LIN {X -0.155,Y -578.900,Z 921.405,A 0.000,B 0.000,C 90.000,E1 108.852} C_DIS
LIN {X -0.107,Y -571.910,Z 921.403,A 0.000,B 0.000,C 90.000,E1 108.471} C_DIS
LIN {X 0.202,Y -564.890,Z 921.401,A 0.000,B 0.000,C 90.000,E1 108.127} C_DIS
LIN {X -0.065,Y -557.655,Z 921.399,A 0.000,B 0.000,C 90.000,E1 107.873} C_DIS
LIN {X -0.326,Y -554.957,Z 921.399,A 0.000,B 0.000,C 90.000,E1 107.764} C_DIS
LIN {X -0.045,Y -553.341,Z 921.398,A 0.000,B 0.000,C 90.000,E1 107.583} C_DIS
LIN {X -0.084,Y -553.320,Z 921.398,A 0.000,B 0.000,C 90.000,E1 107.583} C_DIS
LIN {X 0.080,Y -552.969,Z 921.396,A 0.000,B 0.000,C 90.000,E1 107.347} C_DIS
LIN {X 0.102,Y -553.748,Z 921.385,A 0.000,B 0.000,C 90.000,E1 105.245} C_DIS
LIN {X 0.147,Y -554.848,Z 921.372,A 0.000,B 0.000,C 90.000,E1 103.008} C_DIS
LIN {X -0.166,Y -556.747,Z 921.357,A 0.000,B 0.000,C 90.000,E1 100.254} C_DIS
LIN {X -0.129,Y -557.796,Z 921.349,A 0.000,B 0.000,C 90.000,E1 98.859} C_DIS
LIN {X -0.015,Y -558.994,Z 921.340,A 0.000,B 0.000,C 90.000,E1 97.182} C_DIS
LIN {X -0.155,Y -559.710,Z 921.334,A 0.000,B 0.000,C 90.000,E1 96.087} C_DIS
LIN {X -0.153,Y -560.546,Z 921.326,A 0.000,B 0.000,C 90.000,E1 94.702} C_DIS
LIN {X -0.229,Y -561.254,Z 921.318,A 0.000,B 0.000,C 90.000,E1 93.326} C_DIS
LIN {X -0.283,Y -561.918,Z 921.311,A 0.000,B 0.000,C 90.000,E1 91.949} C_DIS
LIN {X 0.131,Y -562.359,Z 921.305,A 0.000,B 0.000,C 90.000,E1 90.802} C_DIS
LIN {X 0.078,Y -562.761,Z 921.297,A 0.000,B 0.000,C 90.000,E1 89.427} C_DIS
LIN {X -0.075,Y -562.990,Z 921.291,A 0.000,B 0.000,C 90.000,E1 88.339} C_DIS
LIN {X 0.023,Y -563.336,Z 921.282,A 0.000,B 0.000,C 90.000,E1 86.674} C_DIS
LIN {X 0.137,Y -563.594,Z 921.272,A 0.000,B 0.000,C 90.000,E1 85.008} C_DIS
LIN {X -0.167,Y -563.962,Z 921.262,A 0.000,B 0.000,C 90.000,E1 83.109} C_DIS
LIN {X 0.070,Y -564.278,Z 921.253,A 0.000,B 0.000,C 90.000,E1 81.432} C_DIS
LIN {X 0.014,Y -564.989,Z 921.242,A 0.000,B 0.000,C 90.000,E1 79.511} C_DIS
LIN {X -0.025,Y -565.940,Z 921.231,A 0.000,B 0.000,C 90.000,E1 77.589} C_DIS
LIN {X 0.193,Y -567.056,Z 921.220,A 0.000,B 0.000,C 90.000,E1 75.644} C_DIS
LIN {X -0.131,Y -568.000,Z 921.211,A 0.000,B 0.000,C 90.000,E1 74.031} C_DIS
LIN {X 0.112,Y -568.779,Z 921.202,A 0.000,B 0.000,C 90.000,E1 72.362} C_DIS
LIN {X 0.340,Y -569.551,Z 921.191,A 0.000,B 0.000,C 90.000,E1 70.423} C_DIS
LIN {X -0.267,Y -569.891,Z 921.185,A 0.000,B 0.000,C 90.000,E1 69.390} C_DIS
LIN {X 0.036,Y -570.321,Z 921.176,A 0.000,B 0.000,C 90.000,E1 67.720} C_DIS
LIN {X -0.005,Y -570.513,Z 921.169,A 0.000,B 0.000,C 90.000,E1 66.357} C_DIS
LIN {X 0.014,Y -570.742,Z 921.160,A 0.000,B 0.000,C 90.000,E1 64.717} C_DIS
LIN {X 0.198,Y -570.867,Z 921.152,A 0.000,B 0.000,C 90.000,E1 63.332} C_DIS
LIN {X -0.048,Y -570.821,Z 921.143,A 0.000,B 0.000,C 90.000,E1 61.719} C_DIS
LIN {X 0.151,Y -570.814,Z 921.135,A 0.000,B 0.000,C 90.000,E1 60.333} C_DIS
LIN {X 0.036,Y -570.701,Z 921.129,A 0.000,B 0.000,C 90.000,E1 59.253} C_DIS
LIN {X -0.373,Y -570.505,Z 921.123,A 0.000,B 0.000,C 90.000,E1 58.201} C_DIS
LIN {X 0.296,Y -570.066,Z 921.117,A 0.000,B 0.000,C 90.000,E1 57.041} C_DIS
LIN {X 0.167,Y -569.577,Z 921.111,A 0.000,B 0.000,C 90.000,E1 55.960} C_DIS
LIN {X -0.248,Y -569.113,Z 921.107,A 0.000,B 0.000,C 90.000,E1 55.182} C_DIS
LIN {X 0.131,Y -568.532,Z 921.102,A 0.000,B 0.000,C 90.000,E1 54.322} C_DIS
LIN {X 0.171,Y -567.857,Z 921.097,A 0.000,B 0.000,C 90.000,E1 53.497} C_DIS
LIN {X 0.205,Y -566.668,Z 921.091,A 0.000,B 0.000,C 90.000,E1 52.396} C_DIS
LIN {X -0.123,Y -565.340,Z 921.085,A 0.000,B 0.000,C 90.000,E1 51.331} C_DIS
LIN {X 0.235,Y -563.649,Z 921.079,A 0.000,B 0.000,C 90.000,E1 50.194} C_DIS
LIN {X 0.111,Y -562.253,Z 921.074,A 0.000,B 0.000,C 90.000,E1 49.380} C_DIS
LIN {X -0.033,Y -560.643,Z 921.070,A 0.000,B 0.000,C 90.000,E1 48.566} C_DIS
LIN {X 0.176,Y -558.833,Z 921.065,A 0.000,B 0.000,C 90.000,E1 47.715} C_DIS
LIN {X 0.294,Y -557.537,Z 921.062,A 0.000,B 0.000,C 90.000,E1 47.148} C_DIS
LIN {X 0.124,Y -554.396,Z 921.056,A 0.000,B 0.000,C 90.000,E1 46.053} C_DIS
LIN {X -0.220,Y -553.596,Z 921.054,A 0.000,B 0.000,C 90.000,E1 45.810} C_DIS
LIN {X 0.294,Y -550.777,Z 921.050,A 0.000,B 0.000,C 90.000,E1 44.919} C_DIS
LIN {X -0.033,Y -548.775,Z 921.047,A 0.000,B 0.000,C 90.000,E1 44.393} C_DIS
LIN {X 0.042,Y -545.409,Z 921.042,A 0.000,B 0.000,C 90.000,E1 43.542} C_DIS
LIN {X 0.065,Y -543.005,Z 921.039,A 0.000,B 0.000,C 90.000,E1 42.975} C_DIS
LIN {X 0.081,Y -537.557,Z 921.033,A 0.000,B 0.000,C 90.000,E1 41.838} C_DIS
LIN {X -0.142,Y -533.753,Z 921.029,A 0.000,B 0.000,C 90.000,E1 41.148} C_DIS
LIN {X 0.007,Y -529.606,Z 921.025,A 0.000,B 0.000,C 90.000,E1 40.415} C_DIS
LIN {X -0.131,Y -524.206,Z 921.020,A 0.000,B 0.000,C 90.000,E1 39.564} C_DIS
LIN {X 0.068,Y -518.435,Z 921.015,A 0.000,B 0.000,C 90.000,E1 38.669} C_DIS
LIN {X 0.073,Y -513.345,Z 921.011,A 0.000,B 0.000,C 90.000,E1 37.935} C_DIS
LIN {X -0.276,Y -508.013,Z 921.007,A 0.000,B 0.000,C 90.000,E1 37.237} C_DIS
LIN {X 0.134,Y -500.920,Z 921.002,A 0.000,B 0.000,C 90.000,E1 36.297} C_DIS
LIN {X -0.105,Y -495.831,Z 920.998,A 0.000,B 0.000,C 90.000,E1 35.724} C_DIS
LIN {X 0.138,Y -490.507,Z 920.995,A 0.000,B 0.000,C 90.000,E1 35.105} C_DIS
LIN {X 0.216,Y -483.823,Z 920.991,A 0.000,B 0.000,C 90.000,E1 34.405} C_DIS
LIN {X 0.006,Y -477.975,Z 920.988,A 0.000,B 0.000,C 90.000,E1 33.865} C_DIS
LIN {X 0.120,Y -469.147,Z 920.984,A 0.000,B 0.000,C 90.000,E1 33.038} C_DIS
LIN {X -0.025,Y -460.160,Z 920.979,A 0.000,B 0.000,C 90.000,E1 32.260} C_DIS
LIN {X 0.081,Y -447.901,Z 920.974,A 0.000,B 0.000,C 90.000,E1 31.209} C_DIS
LIN {X 0.065,Y -430.957,Z 920.966,A 0.000,B 0.000,C 90.000,E1 29.795} C_DIS
LIN {X 0.023,Y -409.707,Z 920.955,A 0.000,B 0.000,C 90.000,E1 27.897} C_DIS
LIN {X -0.106,Y -401.030,Z 920.950,A 0.000,B 0.000,C 90.000,E1 27.052} C_DIS
LIN {X -0.127,Y -395.925,Z 920.947,A 0.000,B 0.000,C 90.000,E1 26.488} C_DIS
LIN {X -0.007,Y -394.135,Z 920.946,A 0.000,B 0.000,C 90.000,E1 26.232} C_DIS
LIN {X -0.213,Y -392.254,Z 920.944,A 0.000,B 0.000,C 90.000,E1 25.976} C_DIS
LIN {X -0.062,Y -390.731,Z 920.942,A 0.000,B 0.000,C 90.000,E1 25.643} C_DIS
LIN {X -0.113,Y -389.363,Z 920.940,A 0.000,B 0.000,C 90.000,E1 25.155} C_DIS
LIN {X 0.064,Y -388.954,Z 920.939,A 0.000,B 0.000,C 90.000,E1 24.951} C_DIS
LIN {X 0.166,Y -388.518,Z 920.936,A 0.000,B 0.000,C 90.000,E1 24.387} C_DIS
LIN {X 0.058,Y -388.642,Z 920.932,A 0.000,B 0.000,C 90.000,E1 23.695} C_DIS
LIN {X -0.105,Y -392.840,Z 920.906,A 0.000,B 0.000,C 90.000,E1 19.087} C_DIS
LIN {X -0.142,Y -396.197,Z 920.890,A 0.000,B 0.000,C 90.000,E1 16.260} C_DIS
LIN {X 0.067,Y -400.345,Z 920.873,A 0.000,B 0.000,C 90.000,E1 13.063} C_DIS
LIN {X 0.165,Y -404.546,Z 920.857,A 0.000,B 0.000,C 90.000,E1 10.254} C_DIS
LIN {X -0.171,Y -408.566,Z 920.844,A 0.000,B 0.000,C 90.000,E1 7.871} C_DIS
LIN {X -0.138,Y -412.265,Z 920.832,A 0.000,B 0.000,C 90.000,E1 5.796} C_DIS
LIN {X -0.085,Y -415.633,Z 920.823,A 0.000,B 0.000,C 90.000,E1 4.073} C_DIS
LIN {X 0.178,Y -422.235,Z 920.806,A 0.000,B 0.000,C 90.000,E1 0.974} C_DIS
LIN {X 0.034,Y -429.232,Z 920.790,A 0.000,B 0.000,C 90.000,E1 358.108} C_DIS
LIN {X 0.171,Y -431.299,Z 920.786,A 0.000,B 0.000,C 90.000,E1 357.421} C_DIS
LIN {X -0.148,Y -433.347,Z 920.783,A 0.000,B 0.000,C 90.000,E1 356.963} C_DIS
LIN {X -0.112,Y -436.667,Z 920.780,A 0.000,B 0.000,C 90.000,E1 356.445} C_DIS
LIN {X -0.068,Y -438.404,Z 920.779,A 0.000,B 0.000,C 90.000,E1 356.274} C_DIS
LIN {X 0.123,Y -441.542,Z 920.778,A 0.000,B 0.000,C 90.000,E1 355.988} C_DIS
LIN {X 0.114,Y -447.681,Z 920.776,A 0.000,B 0.000,C 90.000,E1 355.641} C_DIS
LIN {X 0.084,Y -456.667,Z 920.774,A 0.000,B 0.000,C 90.000,E1 355.241} C_DIS
LIN {X 0.004,Y -466.607,Z 920.771,A 0.000,B 0.000,C 90.000,E1 354.780} C_DIS
LIN {X 0.197,Y -483.309,Z 920.766,A 0.000,B 0.000,C 90.000,E1 353.913} C_DIS
LIN {X 0.043,Y -493.230,Z 920.763,A 0.000,B 0.000,C 90.000,E1 353.394} C_DIS
LIN {X -0.231,Y -506.078,Z 920.759,A 0.000,B 0.000,C 90.000,E1 352.704} C_DIS
LIN {X -0.105,Y -515.398,Z 920.756,A 0.000,B 0.000,C 90.000,E1 352.129} C_DIS
LIN {X -0.100,Y -521.738,Z 920.754,A 0.000,B 0.000,C 90.000,E1 351.724} C_DIS
LIN {X -0.148,Y -530.798,Z 920.750,A 0.000,B 0.000,C 90.000,E1 351.084} C_DIS
LIN {X -0.007,Y -536.690,Z 920.748,A 0.000,B 0.000,C 90.000,E1 350.622} C_DIS
LIN {X -0.031,Y -544.823,Z 920.744,A 0.000,B 0.000,C 90.000,E1 349.926} C_DIS
LIN {X 0.170,Y -550.298,Z 920.741,A 0.000,B 0.000,C 90.000,E1 349.398} C_DIS
LIN {X 0.037,Y -556.664,Z 920.738,A 0.000,B 0.000,C 90.000,E1 348.757} C_DIS
LIN {X 0.139,Y -564.802,Z 920.732,A 0.000,B 0.000,C 90.000,E1 347.825} C_DIS
LIN {X -0.193,Y -570.375,Z 920.729,A 0.000,B 0.000,C 90.000,E1 347.173} C_DIS
LIN {X 0.286,Y -577.495,Z 920.723,A 0.000,B 0.000,C 90.000,E1 346.172} C_DIS
LIN {X 0.054,Y -582.153,Z 920.720,A 0.000,B 0.000,C 90.000,E1 345.519} C_DIS
LIN {X 0.018,Y -589.016,Z 920.714,A 0.000,B 0.000,C 90.000,E1 344.448} C_DIS
LIN {X 0.142,Y -594.307,Z 920.708,A 0.000,B 0.000,C 90.000,E1 343.504} C_DIS
LIN {X -0.310,Y -600.032,Z 920.703,A 0.000,B 0.000,C 90.000,E1 342.489} C_DIS
LIN {X -0.180,Y -603.379,Z 920.699,A 0.000,B 0.000,C 90.000,E1 341.819} C_DIS
LIN {X 0.250,Y -608.561,Z 920.693,A 0.000,B 0.000,C 90.000,E1 340.732} C_DIS
LIN {X -0.112,Y -611.757,Z 920.690,A 0.000,B 0.000,C 90.000,E1 340.115} C_DIS
LIN {X -0.151,Y -616.431,Z 920.684,A 0.000,B 0.000,C 90.000,E1 339.082} C_DIS
LIN {X 0.094,Y -620.959,Z 920.678,A 0.000,B 0.000,C 90.000,E1 338.028} C_DIS
LIN {X 0.163,Y -626.123,Z 920.671,A 0.000,B 0.000,C 90.000,E1 336.741} C_DIS
LIN {X -0.041,Y -629.861,Z 920.665,A 0.000,B 0.000,C 90.000,E1 335.741} C_DIS
LIN {X 0.147,Y -635.046,Z 920.657,A 0.000,B 0.000,C 90.000,E1 334.204} C_DIS
LIN {X 0.001,Y -637.559,Z 920.653,A 0.000,B 0.000,C 90.000,E1 333.461} C_DIS
LIN {X -0.230,Y -642.060,Z 920.644,A 0.000,B 0.000,C 90.000,E1 331.975} C_DIS
LIN {X -0.139,Y -645.370,Z 920.637,A 0.000,B 0.000,C 90.000,E1 330.717} C_DIS
LIN {X 0.015,Y -648.503,Z 920.630,A 0.000,B 0.000,C 90.000,E1 329.459} C_DIS
LIN {X 0.218,Y -651.364,Z 920.623,A 0.000,B 0.000,C 90.000,E1 328.201} C_DIS
LIN {X -0.187,Y -653.364,Z 920.618,A 0.000,B 0.000,C 90.000,E1 327.248} C_DIS
LIN {X 0.341,Y -655.077,Z 920.613,A 0.000,B 0.000,C 90.000,E1 326.215} C_DIS
LIN {X -0.099,Y -656.881,Z 920.606,A 0.000,B 0.000,C 90.000,E1 325.022} C_DIS
LIN {X 0.023,Y -658.426,Z 920.599,A 0.000,B 0.000,C 90.000,E1 323.783} C_DIS
LIN {X -0.025,Y -659.952,Z 920.591,A 0.000,B 0.000,C 90.000,E1 322.316} C_DIS
LIN {X -0.030,Y -661.230,Z 920.583,A 0.000,B 0.000,C 90.000,E1 320.848} C_DIS
LIN {X -0.018,Y -662.403,Z 920.574,A 0.000,B 0.000,C 90.000,E1 319.380} C_DIS
LIN {X -0.065,Y -664.772,Z 920.561,A 0.000,B 0.000,C 90.000,E1 316.944} C_DIS
LIN {X -0.090,Y -665.637,Z 920.555,A 0.000,B 0.000,C 90.000,E1 315.972} C_DIS
LIN {X -0.093,Y -667.802,Z 920.541,A 0.000,B 0.000,C 90.000,E1 313.299} C_DIS
LIN {X -0.035,Y -669.268,Z 920.532,A 0.000,B 0.000,C 90.000,E1 311.838} C_DIS
LIN {X 0.052,Y -670.558,Z 920.524,A 0.000,B 0.000,C 90.000,E1 310.378} C_DIS
LIN {X -0.280,Y -671.560,Z 920.518,A 0.000,B 0.000,C 90.000,E1 309.197} C_DIS
LIN {X 0.350,Y -672.330,Z 920.512,A 0.000,B 0.000,C 90.000,E1 308.177} C_DIS
LIN {X 0.169,Y -673.343,Z 920.504,A 0.000,B 0.000,C 90.000,E1 306.744} C_DIS
LIN {X 0.005,Y -673.961,Z 920.496,A 0.000,B 0.000,C 90.000,E1 305.311} C_DIS
LIN {X -0.143,Y -674.489,Z 920.490,A 0.000,B 0.000,C 90.000,E1 304.119} C_DIS
LIN {X 0.037,Y -675.372,Z 920.480,A 0.000,B 0.000,C 90.000,E1 302.418} C_DIS
LIN {X -0.170,Y -676.603,Z 920.469,A 0.000,B 0.000,C 90.000,E1 300.512} C_DIS
LIN {X 0.121,Y -680.212,Z 920.451,A 0.000,B 0.000,C 90.000,E1 297.129} C_DIS
LIN {X 0.232,Y -682.979,Z 920.440,A 0.000,B 0.000,C 90.000,E1 295.207} C_DIS
LIN {X 0.163,Y -684.330,Z 920.435,A 0.000,B 0.000,C 90.000,E1 294.259} C_DIS
LIN {X -0.104,Y -685.114,Z 920.431,A 0.000,B 0.000,C 90.000,E1 293.567} C_DIS
LIN {X 0.049,Y -685.476,Z 920.428,A 0.000,B 0.000,C 90.000,E1 293.078} C_DIS
LIN {X 0.210,Y -685.469,Z 920.426,A 0.000,B 0.000,C 90.000,E1 292.589} C_DIS
LIN {X -0.211,Y -685.321,Z 920.424,A 0.000,B 0.000,C 90.000,E1 292.386} C_DIS
LIN {X -0.049,Y -683.903,Z 920.422,A 0.000,B 0.000,C 90.000,E1 291.897} C_DIS
LIN {X -0.097,Y -682.936,Z 920.420,A 0.000,B 0.000,C 90.000,E1 291.663} C_DIS
LIN {X 0.005,Y -682.139,Z 920.420,A 0.000,B 0.000,C 90.000,E1 291.535} C_DIS
LIN {X 0.106,Y -680.957,Z 920.419,A 0.000,B 0.000,C 90.000,E1 291.408} C_DIS
LIN {X 0.061,Y -677.819,Z 920.418,A 0.000,B 0.000,C 90.000,E1 291.173} C_DIS
LIN {X -0.109,Y -676.090,Z 920.417,A 0.000,B 0.000,C 90.000,E1 291.046} C_DIS
LIN {X 0.122,Y -674.544,Z 920.416,A 0.000,B 0.000,C 90.000,E1 290.918} C_DIS
LIN {X -0.114,Y -662.599,Z 920.413,A 0.000,B 0.000,C 90.000,E1 290.301} C_DIS
LIN {X 0.133,Y -661.615,Z 920.412,A 0.000,B 0.000,C 90.000,E1 290.174} C_DIS
LIN {X 0.072,Y -661.583,Z 920.412,A 0.000,B 0.000,C 90.000,E1 290.174} C_DIS
LIN {X -0.280,Y -661.528,Z 920.411,A 0.000,B 0.000,C 90.000,E1 290.066} C_DIS
LIN {X -0.188,Y -661.993,Z 920.410,A 0.000,B 0.000,C 90.000,E1 289.812} C_DIS
LIN {X -0.296,Y -662.586,Z 920.409,A 0.000,B 0.000,C 90.000,E1 289.577} C_DIS
LIN {X -0.224,Y -665.137,Z 920.405,A 0.000,B 0.000,C 90.000,E1 288.960} C_DIS
LIN {X 0.400,Y -671.467,Z 920.399,A 0.000,B 0.000,C 90.000,E1 287.692} C_DIS
LIN {X 0.329,Y -674.341,Z 920.395,A 0.000,B 0.000,C 90.000,E1 287.094} C_DIS
LIN {X 0.158,Y -677.293,Z 920.391,A 0.000,B 0.000,C 90.000,E1 286.386} C_DIS
LIN {X 0.205,Y -679.662,Z 920.387,A 0.000,B 0.000,C 90.000,E1 285.662} C_DIS
LIN {X 0.090,Y -681.503,Z 920.383,A 0.000,B 0.000,C 90.000,E1 284.954} C_DIS
LIN {X -0.004,Y -683.054,Z 920.379,A 0.000,B 0.000,C 90.000,E1 284.245} C_DIS
LIN {X -0.083,Y -684.449,Z 920.375,A 0.000,B 0.000,C 90.000,E1 283.536} C_DIS
LIN {X -0.172,Y -685.879,Z 920.370,A 0.000,B 0.000,C 90.000,E1 282.591} C_DIS
LIN {X -0.213,Y -686.420,Z 920.367,A 0.000,B 0.000,C 90.000,E1 282.119} C_DIS
LIN {X 0.265,Y -687.000,Z 920.363,A 0.000,B 0.000,C 90.000,E1 281.366} C_DIS
LIN {X 0.229,Y -687.135,Z 920.361,A 0.000,B 0.000,C 90.000,E1 280.894} C_DIS
LIN {X 0.209,Y -687.145,Z 920.359,A 0.000,B 0.000,C 90.000,E1 280.658} C_DIS
LIN {X 0.046,Y -686.737,Z 920.357,A 0.000,B 0.000,C 90.000,E1 280.197} C_DIS
LIN {X 0.001,Y -686.012,Z 920.354,A 0.000,B 0.000,C 90.000,E1 279.726} C_DIS
LIN {X -0.139,Y -685.539,Z 920.353,A 0.000,B 0.000,C 90.000,E1 279.500} C_DIS
LIN {X -0.195,Y -684.132,Z 920.350,A 0.000,B 0.000,C 90.000,E1 279.029} C_DIS
LIN {X 0.306,Y -682.261,Z 920.347,A 0.000,B 0.000,C 90.000,E1 278.511} C_DIS
LIN {X 0.124,Y -680.108,Z 920.345,A 0.000,B 0.000,C 90.000,E1 278.049} C_DIS
LIN {X -0.129,Y -676.509,Z 920.341,A 0.000,B 0.000,C 90.000,E1 277.352} C_DIS
LIN {X 0.167,Y -672.653,Z 920.337,A 0.000,B 0.000,C 90.000,E1 276.606} C_DIS
LIN {X 0.004,Y -670.574,Z 920.335,A 0.000,B 0.000,C 90.000,E1 276.258} C_DIS
LIN {X -0.252,Y -667.553,Z 920.332,A 0.000,B 0.000,C 90.000,E1 275.796} C_DIS
LIN {X 0.048,Y -663.220,Z 920.329,A 0.000,B 0.000,C 90.000,E1 275.163} C_DIS
LIN {X -0.257,Y -659.452,Z 920.326,A 0.000,B 0.000,C 90.000,E1 274.702} C_DIS
LIN {X 0.020,Y -655.391,Z 920.323,A 0.000,B 0.000,C 90.000,E1 274.188} C_DIS
LIN {X 0.315,Y -650.942,Z 920.321,A 0.000,B 0.000,C 90.000,E1 273.669} C_DIS
LIN {X -0.068,Y -644.753,Z 920.317,A 0.000,B 0.000,C 90.000,E1 273.094} C_DIS
LIN {X -0.155,Y -638.118,Z 920.314,A 0.000,B 0.000,C 90.000,E1 272.522} C_DIS
LIN {X 0.081,Y -631.037,Z 920.311,A 0.000,B 0.000,C 90.000,E1 271.949} C_DIS
LIN {X 0.129,Y -623.512,Z 920.308,A 0.000,B 0.000,C 90.000,E1 271.432} C_DIS
LIN {X 0.290,Y -617.281,Z 920.306,A 0.000,B 0.000,C 90.000,E1 271.031} C_DIS
LIN {X 0.015,Y -610.854,Z 920.304,A 0.000,B 0.000,C 90.000,E1 270.688} C_DIS
LIN {X -0.274,Y -602.351,Z 920.302,A 0.000,B 0.000,C 90.000,E1 270.286} C_DIS
LIN {X 0.237,Y -597.258,Z 920.300,A 0.000,B 0.000,C 90.000,E1 270.000} C_DIS
LIN {X 0.209,Y -589.987,Z 920.299,A 0.000,B 0.000,C 90.000,E1 269.714} C_DIS
LIN {X 0.037,Y -584.694,Z 920.298,A 0.000,B 0.000,C 90.000,E1 269.542} C_DIS
LIN {X 0.157,Y -577.196,Z 920.296,A 0.000,B 0.000,C 90.000,E1 269.312} C_DIS
LIN {X -0.029,Y -571.343,Z 920.296,A 0.000,B 0.000,C 90.000,E1 269.198} C_DIS
LIN {X -0.021,Y -564.836,Z 920.295,A 0.000,B 0.000,C 90.000,E1 269.083} C_DIS
LIN {X -0.204,Y -557.307,Z 920.294,A 0.000,B 0.000,C 90.000,E1 269.026} C_DIS
LIN {X -0.039,Y -552.254,Z 920.294,A 0.000,B 0.000,C 90.000,E1 268.969} C_DIS
LIN {X 0.174,Y -549.119,Z 920.294,A 0.000,B 0.000,C 90.000,E1 268.854} C_DIS
LIN {X 0.199,Y -548.084,Z 920.293,A 0.000,B 0.000,C 90.000,E1 268.797} C_DIS
LIN {X -0.230,Y -546.605,Z 920.293,A 0.000,B 0.000,C 90.000,E1 268.740} C_DIS
LIN {X -0.237,Y -545.167,Z 920.292,A 0.000,B 0.000,C 90.000,E1 268.568} C_DIS
LIN {X -0.070,Y -544.408,Z 920.291,A 0.000,B 0.000,C 90.000,E1 268.339} C_DIS
LIN {X -0.120,Y -543.475,Z 920.288,A 0.000,B 0.000,C 90.000,E1 267.879} C_DIS
LIN {X -0.233,Y -540.172,Z 920.268,A 0.000,B 0.000,C 90.000,E1 264.204} C_DIS
LIN {X -0.103,Y -539.375,Z 920.261,A 0.000,B 0.000,C 90.000,E1 263.053} C_DIS
LIN {X 0.147,Y -538.302,Z 920.253,A 0.000,B 0.000,C 90.000,E1 261.602} C_DIS
LIN {X -0.210,Y -537.310,Z 920.247,A 0.000,B 0.000,C 90.000,E1 260.500} C_DIS
LIN {X -0.056,Y -536.131,Z 920.241,A 0.000,B 0.000,C 90.000,E1 259.342} C_DIS
LIN {X 0.172,Y -534.643,Z 920.234,A 0.000,B 0.000,C 90.000,E1 258.173} C_DIS
LIN {X 0.023,Y -532.888,Z 920.227,A 0.000,B 0.000,C 90.000,E1 256.756} C_DIS
LIN {X -0.111,Y -530.764,Z 920.217,A 0.000,B 0.000,C 90.000,E1 255.046} C_DIS
LIN {X -0.161,Y -528.629,Z 920.207,A 0.000,B 0.000,C 90.000,E1 253.323} C_DIS
LIN {X 0.212,Y -527.254,Z 920.201,A 0.000,B 0.000,C 90.000,E1 252.127} C_DIS
LIN {X 0.051,Y -524.234,Z 920.188,A 0.000,B 0.000,C 90.000,E1 249.826} C_DIS
LIN {X -0.305,Y -522.326,Z 920.180,A 0.000,B 0.000,C 90.000,E1 248.411} C_DIS
LIN {X -0.163,Y -520.751,Z 920.173,A 0.000,B 0.000,C 90.000,E1 247.230} C_DIS
LIN {X -0.046,Y -519.075,Z 920.167,A 0.000,B 0.000,C 90.000,E1 246.049} C_DIS
LIN {X -0.077,Y -516.796,Z 920.159,A 0.000,B 0.000,C 90.000,E1 244.588} C_DIS
LIN {X 0.194,Y -515.032,Z 920.152,A 0.000,B 0.000,C 90.000,E1 243.384} C_DIS
LIN {X -0.030,Y -512.132,Z 920.142,A 0.000,B 0.000,C 90.000,E1 241.641} C_DIS
LIN {X -0.053,Y -510.025,Z 920.136,A 0.000,B 0.000,C 90.000,E1 240.461} C_DIS
LIN {X -0.218,Y -507.339,Z 920.128,A 0.000,B 0.000,C 90.000,E1 238.997} C_DIS
LIN {X 0.056,Y -505.700,Z 920.123,A 0.000,B 0.000,C 90.000,E1 238.074} C_DIS
LIN {X 0.150,Y -503.937,Z 920.118,A 0.000,B 0.000,C 90.000,E1 237.168} C_DIS
LIN {X -0.047,Y -501.987,Z 920.113,A 0.000,B 0.000,C 90.000,E1 236.294} C_DIS
LIN {X 0.046,Y -497.955,Z 920.103,A 0.000,B 0.000,C 90.000,E1 234.482} C_DIS
LIN {X 0.190,Y -493.268,Z 920.091,A 0.000,B 0.000,C 90.000,E1 232.351} C_DIS
LIN {X -0.254,Y -489.932,Z 920.083,A 0.000,B 0.000,C 90.000,E1 230.884} C_DIS
LIN {X 0.070,Y -485.783,Z 920.072,A 0.000,B 0.000,C 90.000,E1 229.013} C_DIS
LIN {X 0.254,Y -481.684,Z 920.062,A 0.000,B 0.000,C 90.000,E1 227.148} C_DIS
LIN {X -0.123,Y -478.298,Z 920.054,A 0.000,B 0.000,C 90.000,E1 225.648} C_DIS
LIN {X -0.002,Y -475.535,Z 920.047,A 0.000,B 0.000,C 90.000,E1 224.393} C_DIS
LIN {X -0.059,Y -471.328,Z 920.036,A 0.000,B 0.000,C 90.000,E1 222.528} C_DIS
LIN {X 0.075,Y -467.743,Z 920.028,A 0.000,B 0.000,C 90.000,E1 220.943} C_DIS
LIN {X -0.100,Y -463.720,Z 920.017,A 0.000,B 0.000,C 90.000,E1 219.072} C_DIS
LIN {X -0.151,Y -461.096,Z 920.010,A 0.000,B 0.000,C 90.000,E1 217.810} C_DIS
LIN {X -0.149,Y -457.641,Z 920.001,A 0.000,B 0.000,C 90.000,E1 216.217} C_DIS
LIN {X -0.114,Y -454.260,Z 919.992,A 0.000,B 0.000,C 90.000,E1 214.612} C_DIS
LIN {X 0.050,Y -452.149,Z 919.987,A 0.000,B 0.000,C 90.000,E1 213.627} C_DIS
LIN {X -0.126,Y -447.099,Z 919.974,A 0.000,B 0.000,C 90.000,E1 211.386} C_DIS
LIN {X -0.077,Y -444.231,Z 919.967,A 0.000,B 0.000,C 90.000,E1 210.079} C_DIS
LIN {X 0.032,Y -439.969,Z 919.956,A 0.000,B 0.000,C 90.000,E1 208.103} C_DIS
LIN {X 0.213,Y -435.640,Z 919.945,A 0.000,B 0.000,C 90.000,E1 206.104} C_DIS
LIN {X -0.095,Y -430.535,Z 919.932,A 0.000,B 0.000,C 90.000,E1 203.823} C_DIS
LIN {X 0.111,Y -426.182,Z 919.921,A 0.000,B 0.000,C 90.000,E1 201.791} C_DIS
LIN {X -0.003,Y -421.085,Z 919.908,A 0.000,B 0.000,C 90.000,E1 199.450} C_DIS
LIN {X 0.091,Y -417.144,Z 919.897,A 0.000,B 0.000,C 90.000,E1 197.402} C_DIS
LIN {X -0.061,Y -413.750,Z 919.887,A 0.000,B 0.000,C 90.000,E1 195.717} C_DIS
LIN {X 0.038,Y -408.861,Z 919.874,A 0.000,B 0.000,C 90.000,E1 193.300} C_DIS
LIN {X -0.102,Y -405.392,Z 919.864,A 0.000,B 0.000,C 90.000,E1 191.591} C_DIS
LIN {X -0.079,Y -401.278,Z 919.853,A 0.000,B 0.000,C 90.000,E1 189.500} C_DIS
LIN {X -0.154,Y -397.122,Z 919.841,A 0.000,B 0.000,C 90.000,E1 187.409} C_DIS
LIN {X -0.176,Y -391.702,Z 919.825,A 0.000,B 0.000,C 90.000,E1 184.588} C_DIS
LIN {X 0.130,Y -387.977,Z 919.814,A 0.000,B 0.000,C 90.000,E1 182.407} C_DIS
LIN {X -0.161,Y -383.793,Z 919.800,A 0.000,B 0.000,C 90.000,E1 179.943} C_DIS
LIN {X -0.032,Y -379.438,Z 919.782,A 0.000,B 0.000,C 90.000,E1 176.674} C_DIS
LIN {X -0.154,Y -378.609,Z 919.773,A 0.000,B 0.000,C 90.000,E1 175.241} C_DIS
LIN {X 0.015,Y -378.856,Z 919.769,A 0.000,B 0.000,C 90.000,E1 174.489} C_DIS
LIN {X -0.125,Y -379.208,Z 919.767,A 0.000,B 0.000,C 90.000,E1 174.147} C_DIS
LIN {X 0.152,Y -379.733,Z 919.765,A 0.000,B 0.000,C 90.000,E1 173.742} C_DIS
LIN {X -0.017,Y -381.035,Z 919.762,A 0.000,B 0.000,C 90.000,E1 173.223} C_DIS
LIN {X -0.026,Y -382.589,Z 919.760,A 0.000,B 0.000,C 90.000,E1 172.818} C_DIS
LIN {X -0.113,Y -384.408,Z 919.758,A 0.000,B 0.000,C 90.000,E1 172.470} C_DIS
LIN {X -0.180,Y -385.433,Z 919.757,A 0.000,B 0.000,C 90.000,E1 172.299} C_DIS
LIN {X 0.026,Y -391.627,Z 919.753,A 0.000,B 0.000,C 90.000,E1 171.546} C_DIS
LIN {X 0.158,Y -397.375,Z 919.750,A 0.000,B 0.000,C 90.000,E1 171.027} C_DIS
LIN {X 0.179,Y -410.907,Z 919.745,A 0.000,B 0.000,C 90.000,E1 170.038} C_DIS
LIN {X 0.002,Y -417.361,Z 919.742,A 0.000,B 0.000,C 90.000,E1 169.634} C_DIS
LIN {X 0.124,Y -426.783,Z 919.739,A 0.000,B 0.000,C 90.000,E1 168.926} C_DIS
LIN {X -0.092,Y -433.196,Z 919.736,A 0.000,B 0.000,C 90.000,E1 168.465} C_DIS
LIN {X -0.054,Y -442.292,Z 919.732,A 0.000,B 0.000,C 90.000,E1 167.701} C_DIS
LIN {X -0.061,Y -448.369,Z 919.729,A 0.000,B 0.000,C 90.000,E1 167.173} C_DIS
LIN {X 0.066,Y -460.184,Z 919.723,A 0.000,B 0.000,C 90.000,E1 166.061} C_DIS
LIN {X -0.106,Y -465.604,Z 919.720,A 0.000,B 0.000,C 90.000,E1 165.519} C_DIS
LIN {X 0.220,Y -473.673,Z 919.715,A 0.000,B 0.000,C 90.000,E1 164.629} C_DIS
LIN {X 0.228,Y -482.964,Z 919.709,A 0.000,B 0.000,C 90.000,E1 163.559} C_DIS
LIN {X -0.228,Y -491.555,Z 919.703,A 0.000,B 0.000,C 90.000,E1 162.543} C_DIS
LIN {X 0.046,Y -501.669,Z 919.695,A 0.000,B 0.000,C 90.000,E1 161.148} C_DIS
LIN {X -0.154,Y -511.091,Z 919.688,A 0.000,B 0.000,C 90.000,E1 159.826} C_DIS
LIN {X 0.194,Y -517.237,Z 919.683,A 0.000,B 0.000,C 90.000,E1 158.901} C_DIS
LIN {X -0.230,Y -526.718,Z 919.675,A 0.000,B 0.000,C 90.000,E1 157.486} C_DIS
LIN {X 0.003,Y -534.000,Z 919.668,A 0.000,B 0.000,C 90.000,E1 156.305} C_DIS
LIN {X -0.025,Y -541.956,Z 919.661,A 0.000,B 0.000,C 90.000,E1 155.025} C_DIS
LIN {X -0.180,Y -546.209,Z 919.657,A 0.000,B 0.000,C 90.000,E1 154.332} C_DIS
LIN {X 0.085,Y -552.668,Z 919.651,A 0.000,B 0.000,C 90.000,E1 153.179} C_DIS
LIN {X 0.128,Y -555.767,Z 919.648,A 0.000,B 0.000,C 90.000,E1 152.615} C_DIS
LIN {X 0.032,Y -561.654,Z 919.642,A 0.000,B 0.000,C 90.000,E1 151.513} C_DIS
LIN {X 0.014,Y -567.161,Z 919.636,A 0.000,B 0.000,C 90.000,E1 150.411} C_DIS
LIN {X -0.139,Y -572.374,Z 919.630,A 0.000,B 0.000,C 90.000,E1 149.331} C_DIS
LIN {X 0.265,Y -579.794,Z 919.621,A 0.000,B 0.000,C 90.000,E1 147.661} C_DIS
LIN {X -0.171,Y -586.639,Z 919.612,A 0.000,B 0.000,C 90.000,E1 146.087} C_DIS
LIN {X -0.008,Y -592.209,Z 919.604,A 0.000,B 0.000,C 90.000,E1 144.736} C_DIS
LIN {X -0.091,Y -597.354,Z 919.597,A 0.000,B 0.000,C 90.000,E1 143.417} C_DIS
LIN {X 0.014,Y -601.341,Z 919.591,A 0.000,B 0.000,C 90.000,E1 142.351} C_DIS
LIN {X 0.082,Y -610.622,Z 919.578,A 0.000,B 0.000,C 90.000,E1 139.989} C_DIS
LIN {X 0.231,Y -617.886,Z 919.568,A 0.000,B 0.000,C 90.000,E1 138.162} C_DIS
LIN {X 0.090,Y -625.194,Z 919.558,A 0.000,B 0.000,C 90.000,E1 136.377} C_DIS
LIN {X -0.308,Y -628.455,Z 919.553,A 0.000,B 0.000,C 90.000,E1 135.648} C_DIS
LIN {X -0.008,Y -633.570,Z 919.546,A 0.000,B 0.000,C 90.000,E1 134.352} C_DIS
LIN {X -0.061,Y -638.658,Z 919.539,A 0.000,B 0.000,C 90.000,E1 133.095} C_DIS
LIN {X -0.030,Y -643.619,Z 919.532,A 0.000,B 0.000,C 90.000,E1 131.838} C_DIS
LIN {X 0.073,Y -649.552,Z 919.524,A 0.000,B 0.000,C 90.000,E1 130.334} C_DIS
LIN {X -0.156,Y -654.308,Z 919.517,A 0.000,B 0.000,C 90.000,E1 129.116} C_DIS
LIN {X -0.216,Y -659.049,Z 919.510,A 0.000,B 0.000,C 90.000,E1 127.890} C_DIS
LIN {X -0.194,Y -663.606,Z 919.504,A 0.000,B 0.000,C 90.000,E1 126.664} C_DIS
LIN {X -0.176,Y -666.306,Z 919.500,A 0.000,B 0.000,C 90.000,E1 125.931} C_DIS
LIN {X 0.112,Y -670.594,Z 919.493,A 0.000,B 0.000,C 90.000,E1 124.692} C_DIS
LIN {X -0.196,Y -673.042,Z 919.489,A 0.000,B 0.000,C 90.000,E1 123.992} C_DIS
LIN {X 0.079,Y -675.248,Z 919.485,A 0.000,B 0.000,C 90.000,E1 123.245} C_DIS
LIN {X -0.016,Y -678.014,Z 919.479,A 0.000,B 0.000,C 90.000,E1 122.291} C_DIS
LIN {X -0.267,Y -679.859,Z 919.475,A 0.000,B 0.000,C 90.000,E1 121.592} C_DIS
LIN {X -0.123,Y -682.536,Z 919.469,A 0.000,B 0.000,C 90.000,E1 120.384} C_DIS
LIN {X -0.104,Y -683.929,Z 919.465,A 0.000,B 0.000,C 90.000,E1 119.667} C_DIS
LIN {X -0.237,Y -685.877,Z 919.458,A 0.000,B 0.000,C 90.000,E1 118.487} C_DIS
LIN {X 0.202,Y -686.577,Z 919.456,A 0.000,B 0.000,C 90.000,E1 117.975} C_DIS
LIN {X -0.123,Y -687.474,Z 919.450,A 0.000,B 0.000,C 90.000,E1 117.052} C_DIS
LIN {X -0.139,Y -687.906,Z 919.445,A 0.000,B 0.000,C 90.000,E1 116.104} C_DIS
LIN {X -0.143,Y -688.081,Z 919.440,A 0.000,B 0.000,C 90.000,E1 115.155} C_DIS
LIN {X -0.372,Y -688.008,Z 919.436,A 0.000,B 0.000,C 90.000,E1 114.463} C_DIS
LIN {X 0.081,Y -687.786,Z 919.433,A 0.000,B 0.000,C 90.000,E1 113.951} C_DIS
LIN {X 0.254,Y -687.339,Z 919.431,A 0.000,B 0.000,C 90.000,E1 113.462} C_DIS
LIN {X -0.203,Y -686.389,Z 919.428,A 0.000,B 0.000,C 90.000,E1 113.025} C_DIS
LIN {X 0.017,Y -685.439,Z 919.427,A 0.000,B 0.000,C 90.000,E1 112.770} C_DIS
LIN {X 0.179,Y -682.597,Z 919.424,A 0.000,B 0.000,C 90.000,E1 112.280} C_DIS
LIN {X 0.281,Y -681.629,Z 919.423,A 0.000,B 0.000,C 90.000,E1 112.153} C_DIS
LIN {X -0.248,Y -680.163,Z 919.423,A 0.000,B 0.000,C 90.000,E1 112.078} C_DIS
LIN {X -0.014,Y -678.333,Z 919.422,A 0.000,B 0.000,C 90.000,E1 111.950} C_DIS
LIN {X 0.240,Y -671.063,Z 919.420,A 0.000,B 0.000,C 90.000,E1 111.589} C_DIS
LIN {X -0.024,Y -668.667,Z 919.420,A 0.000,B 0.000,C 90.000,E1 111.535} C_DIS
LIN {X -0.116,Y -664.292,Z 919.419,A 0.000,B 0.000,C 90.000,E1 111.461} C_DIS
LIN {X -0.094,Y -660.278,Z 919.419,A 0.000,B 0.000,C 90.000,E1 111.408} C_DIS
LIN {X -0.006,Y -649.933,Z 919.419,A 0.000,B 0.000,C 90.000,E1 111.354} C_DIS
LIN {X -0.244,Y -641.800,Z 919.419,A 0.000,B 0.000,C 90.000,E1 111.354} C_DIS
LIN {X -0.027,Y -636.274,Z 919.418,A 0.000,B 0.000,C 90.000,E1 111.280} C_DIS
LIN {X 0.026,Y -628.250,Z 919.418,A 0.000,B 0.000,C 90.000,E1 111.153} C_DIS
LIN {X 0.266,Y -621.108,Z 919.417,A 0.000,B 0.000,C 90.000,E1 110.972} C_DIS
LIN {X -0.180,Y -613.710,Z 919.415,A 0.000,B 0.000,C 90.000,E1 110.791} C_DIS
LIN {X 0.016,Y -605.227,Z 919.414,A 0.000,B 0.000,C 90.000,E1 110.429} C_DIS
LIN {X 0.179,Y -598.424,Z 919.412,A 0.000,B 0.000,C 90.000,E1 110.066} C_DIS
LIN {X -0.059,Y -580.283,Z 919.405,A 0.000,B 0.000,C 90.000,E1 108.906} C_DIS
LIN {X 0.127,Y -575.121,Z 919.403,A 0.000,B 0.000,C 90.000,E1 108.598} C_DIS
LIN {X -0.058,Y -569.946,Z 919.402,A 0.000,B 0.000,C 90.000,E1 108.362} C_DIS
LIN {X 0.009,Y -564.660,Z 919.401,A 0.000,B 0.000,C 90.000,E1 108.127} C_DIS
LIN {X -0.236,Y -557.508,Z 919.399,A 0.000,B 0.000,C 90.000,E1 107.873} C_DIS
LIN {X -0.148,Y -555.446,Z 919.399,A 0.000,B 0.000,C 90.000,E1 107.764} C_DIS
LIN {X -0.072,Y -553.512,Z 919.398,A 0.000,B 0.000,C 90.000,E1 107.583} C_DIS
LIN {X -0.109,Y -553.490,Z 919.398,A 0.000,B 0.000,C 90.000,E1 107.583} C_DIS
LIN {X 0.115,Y -553.216,Z 919.396,A 0.000,B 0.000,C 90.000,E1 107.330} C_DIS
LIN {X 0.227,Y -553.456,Z 919.391,A 0.000,B 0.000,C 90.000,E1 106.315} C_DIS
LIN {X -0.111,Y -554.052,Z 919.383,A 0.000,B 0.000,C 90.000,E1 104.954} C_DIS
LIN {X 0.198,Y -555.353,Z 919.369,A 0.000,B 0.000,C 90.000,E1 102.411} C_DIS
LIN {X 0.059,Y -556.928,Z 919.357,A 0.000,B 0.000,C 90.000,E1 100.197} C_DIS
LIN {X 0.103,Y -557.976,Z 919.349,A 0.000,B 0.000,C 90.000,E1 98.803} C_DIS
LIN {X 0.223,Y -559.176,Z 919.340,A 0.000,B 0.000,C 90.000,E1 97.125} C_DIS
LIN {X 0.087,Y -559.855,Z 919.334,A 0.000,B 0.000,C 90.000,E1 96.030} C_DIS
LIN {X 0.093,Y -560.687,Z 919.326,A 0.000,B 0.000,C 90.000,E1 94.645} C_DIS
LIN {X 0.145,Y -561.517,Z 919.317,A 0.000,B 0.000,C 90.000,E1 92.980} C_DIS
LIN {X 0.086,Y -562.143,Z 919.309,A 0.000,B 0.000,C 90.000,E1 91.604} C_DIS
LIN {X -0.075,Y -562.561,Z 919.303,A 0.000,B 0.000,C 90.000,E1 90.516} C_DIS
LIN {X -0.227,Y -562.854,Z 919.297,A 0.000,B 0.000,C 90.000,E1 89.427} C_DIS
LIN {X -0.258,Y -563.138,Z 919.289,A 0.000,B 0.000,C 90.000,E1 88.051} C_DIS
LIN {X 0.283,Y -563.427,Z 919.281,A 0.000,B 0.000,C 90.000,E1 86.617} C_DIS
LIN {X 0.254,Y -563.655,Z 919.274,A 0.000,B 0.000,C 90.000,E1 85.241} C_DIS
LIN {X 0.007,Y -563.987,Z 919.263,A 0.000,B 0.000,C 90.000,E1 83.337} C_DIS
LIN {X 0.253,Y -564.326,Z 919.254,A 0.000,B 0.000,C 90.000,E1 81.659} C_DIS
LIN {X 0.109,Y -564.981,Z 919.243,A 0.000,B 0.000,C 90.000,E1 79.746} C_DIS
LIN {X 0.067,Y -565.897,Z 919.232,A 0.000,B 0.000,C 90.000,E1 77.825} C_DIS
LIN {X -0.268,Y -567.008,Z 919.222,A 0.000,B 0.000,C 90.000,E1 75.936} C_DIS
LIN {X 0.180,Y -567.775,Z 919.214,A 0.000,B 0.000,C 90.000,E1 74.519} C_DIS
LIN {X -0.083,Y -568.349,Z 919.208,A 0.000,B 0.000,C 90.000,E1 73.449} C_DIS
LIN {X 0.164,Y -568.971,Z 919.200,A 0.000,B 0.000,C 90.000,E1 72.054} C_DIS
LIN {X -0.327,Y -569.704,Z 919.190,A 0.000,B 0.000,C 90.000,E1 70.188} C_DIS
LIN {X 0.147,Y -570.062,Z 919.182,A 0.000,B 0.000,C 90.000,E1 68.773} C_DIS
LIN {X 0.278,Y -570.326,Z 919.176,A 0.000,B 0.000,C 90.000,E1 67.667} C_DIS
LIN {X -0.117,Y -570.502,Z 919.170,A 0.000,B 0.000,C 90.000,E1 66.613} C_DIS
LIN {X 0.245,Y -570.741,Z 919.159,A 0.000,B 0.000,C 90.000,E1 64.665} C_DIS
LIN {X 0.003,Y -570.809,Z 919.150,A 0.000,B 0.000,C 90.000,E1 63.050} C_DIS
LIN {X -0.061,Y -570.789,Z 919.143,A 0.000,B 0.000,C 90.000,E1 61.691} C_DIS
LIN {X -0.134,Y -570.773,Z 919.135,A 0.000,B 0.000,C 90.000,E1 60.333} C_DIS
LIN {X 0.240,Y -570.637,Z 919.129,A 0.000,B 0.000,C 90.000,E1 59.203} C_DIS
LIN {X 0.005,Y -570.541,Z 919.125,A 0.000,B 0.000,C 90.000,E1 58.408} C_DIS
LIN {X 0.009,Y -569.969,Z 919.117,A 0.000,B 0.000,C 90.000,E1 57.041} C_DIS
LIN {X 0.002,Y -569.306,Z 919.109,A 0.000,B 0.000,C 90.000,E1 55.674} C_DIS
LIN {X 0.178,Y -568.617,Z 919.103,A 0.000,B 0.000,C 90.000,E1 54.562} C_DIS
LIN {X -0.122,Y -567.658,Z 919.097,A 0.000,B 0.000,C 90.000,E1 53.497} C_DIS
LIN {X -0.090,Y -566.451,Z 919.091,A 0.000,B 0.000,C 90.000,E1 52.396} C_DIS
LIN {X -0.067,Y -565.096,Z 919.085,A 0.000,B 0.000,C 90.000,E1 51.295} C_DIS
LIN {X -0.065,Y -563.362,Z 919.079,A 0.000,B 0.000,C 90.000,E1 50.194} C_DIS
LIN {X -0.191,Y -561.930,Z 919.074,A 0.000,B 0.000,C 90.000,E1 49.380} C_DIS
LIN {X -0.004,Y -560.904,Z 919.071,A 0.000,B 0.000,C 90.000,E1 48.809} C_DIS
LIN {X -0.132,Y -558.431,Z 919.065,A 0.000,B 0.000,C 90.000,E1 47.715} C_DIS
LIN {X -0.016,Y -557.093,Z 919.062,A 0.000,B 0.000,C 90.000,E1 47.148} C_DIS
LIN {X 0.155,Y -554.731,Z 919.057,A 0.000,B 0.000,C 90.000,E1 46.296} C_DIS
LIN {X 0.248,Y -553.062,Z 919.054,A 0.000,B 0.000,C 90.000,E1 45.729} C_DIS
LIN {X -0.025,Y -550.179,Z 919.050,A 0.000,B 0.000,C 90.000,E1 44.919} C_DIS
LIN {X -0.324,Y -547.012,Z 919.045,A 0.000,B 0.000,C 90.000,E1 44.109} C_DIS
LIN {X -0.285,Y -544.716,Z 919.042,A 0.000,B 0.000,C 90.000,E1 43.542} C_DIS
LIN {X -0.064,Y -542.926,Z 919.039,A 0.000,B 0.000,C 90.000,E1 43.095} C_DIS
LIN {X -0.259,Y -536.716,Z 919.032,A 0.000,B 0.000,C 90.000,E1 41.838} C_DIS
LIN {X 0.265,Y -532.853,Z 919.028,A 0.000,B 0.000,C 90.000,E1 41.067} C_DIS
LIN {X -0.164,Y -529.519,Z 919.025,A 0.000,B 0.000,C 90.000,E1 40.539} C_DIS
LIN {X -0.052,Y -525.018,Z 919.021,A 0.000,B 0.000,C 90.000,E1 39.806} C_DIS
LIN {X 0.160,Y -519.322,Z 919.016,A 0.000,B 0.000,C 90.000,E1 38.910} C_DIS
LIN {X 0.175,Y -514.228,Z 919.012,A 0.000,B 0.000,C 90.000,E1 38.177} C_DIS
LIN {X 0.144,Y -508.876,Z 919.008,A 0.000,B 0.000,C 90.000,E1 37.443} C_DIS
LIN {X -0.040,Y -504.280,Z 919.005,A 0.000,B 0.000,C 90.000,E1 36.870} C_DIS
LIN {X 0.235,Y -498.169,Z 919.001,A 0.000,B 0.000,C 90.000,E1 36.091} C_DIS
LIN {X 0.006,Y -492.866,Z 918.997,A 0.000,B 0.000,C 90.000,E1 35.518} C_DIS
LIN {X -0.248,Y -488.801,Z 918.995,A 0.000,B 0.000,C 90.000,E1 35.105} C_DIS
LIN {X 0.169,Y -483.174,Z 918.992,A 0.000,B 0.000,C 90.000,E1 34.485} C_DIS
LIN {X 0.304,Y -477.362,Z 918.989,A 0.000,B 0.000,C 90.000,E1 33.913} C_DIS
LIN {X 0.002,Y -467.053,Z 918.983,A 0.000,B 0.000,C 90.000,E1 33.007} C_DIS
LIN {X 0.061,Y -461.011,Z 918.980,A 0.000,B 0.000,C 90.000,E1 32.467} C_DIS
LIN {X -0.184,Y -447.281,Z 918.974,A 0.000,B 0.000,C 90.000,E1 31.337} C_DIS
LIN {X 0.211,Y -431.855,Z 918.967,A 0.000,B 0.000,C 90.000,E1 30.001} C_DIS
LIN {X -0.101,Y -412.031,Z 918.957,A 0.000,B 0.000,C 90.000,E1 28.281} C_DIS
LIN {X -0.117,Y -400.200,Z 918.951,A 0.000,B 0.000,C 90.000,E1 27.129} C_DIS
LIN {X 0.138,Y -396.030,Z 918.948,A 0.000,B 0.000,C 90.000,E1 26.616} C_DIS
LIN {X 0.199,Y -392.507,Z 918.945,A 0.000,B 0.000,C 90.000,E1 26.104} C_DIS
LIN {X -0.201,Y -390.428,Z 918.943,A 0.000,B 0.000,C 90.000,E1 25.720} C_DIS
LIN {X -0.031,Y -389.145,Z 918.940,A 0.000,B 0.000,C 90.000,E1 25.155} C_DIS
LIN {X -0.173,Y -388.538,Z 918.936,A 0.000,B 0.000,C 90.000,E1 24.463} C_DIS
LIN {X 0.078,Y -388.705,Z 918.932,A 0.000,B 0.000,C 90.000,E1 23.718} C_DIS
LIN {X 0.027,Y -392.569,Z 918.908,A 0.000,B 0.000,C 90.000,E1 19.450} C_DIS
LIN {X 0.046,Y -396.307,Z 918.890,A 0.000,B 0.000,C 90.000,E1 16.260} C_DIS
LIN {X -0.129,Y -400.450,Z 918.873,A 0.000,B 0.000,C 90.000,E1 13.119} C_DIS
LIN {X -0.033,Y -404.100,Z 918.859,A 0.000,B 0.000,C 90.000,E1 10.658} C_DIS
LIN {X 0.033,Y -408.659,Z 918.844,A 0.000,B 0.000,C 90.000,E1 7.871} C_DIS
LIN {X 0.069,Y -412.333,Z 918.832,A 0.000,B 0.000,C 90.000,E1 5.796} C_DIS
LIN {X 0.174,Y -417.087,Z 918.819,A 0.000,B 0.000,C 90.000,E1 3.383} C_DIS
LIN {X 0.054,Y -423.833,Z 918.802,A 0.000,B 0.000,C 90.000,E1 0.344} C_DIS
LIN {X 0.104,Y -430.265,Z 918.788,A 0.000,B 0.000,C 90.000,E1 357.764} C_DIS
LIN {X 0.212,Y -431.926,Z 918.785,A 0.000,B 0.000,C 90.000,E1 357.249} C_DIS
LIN {X -0.082,Y -434.116,Z 918.782,A 0.000,B 0.000,C 90.000,E1 356.788} C_DIS
LIN {X -0.076,Y -437.074,Z 918.780,A 0.000,B 0.000,C 90.000,E1 356.331} C_DIS
LIN {X -0.110,Y -442.669,Z 918.777,A 0.000,B 0.000,C 90.000,E1 355.869} C_DIS
LIN {X -0.147,Y -447.940,Z 918.775,A 0.000,B 0.000,C 90.000,E1 355.584} C_DIS
LIN {X -0.128,Y -456.948,Z 918.773,A 0.000,B 0.000,C 90.000,E1 355.179} C_DIS
LIN {X 0.115,Y -467.137,Z 918.771,A 0.000,B 0.000,C 90.000,E1 354.666} C_DIS
LIN {X -0.197,Y -480.538,Z 918.767,A 0.000,B 0.000,C 90.000,E1 354.033} C_DIS
LIN {X -0.016,Y -491.970,Z 918.763,A 0.000,B 0.000,C 90.000,E1 353.394} C_DIS
LIN {X -0.132,Y -503.547,Z 918.760,A 0.000,B 0.000,C 90.000,E1 352.761} C_DIS
LIN {X -0.064,Y -513.252,Z 918.757,A 0.000,B 0.000,C 90.000,E1 352.186} C_DIS
LIN {X 0.179,Y -521.161,Z 918.754,A 0.000,B 0.000,C 90.000,E1 351.659} C_DIS
LIN {X 0.051,Y -530.244,Z 918.750,A 0.000,B 0.000,C 90.000,E1 351.027} C_DIS
LIN {X 0.210,Y -536.221,Z 918.748,A 0.000,B 0.000,C 90.000,E1 350.566} C_DIS
LIN {X 0.098,Y -543.218,Z 918.744,A 0.000,B 0.000,C 90.000,E1 349.982} C_DIS
LIN {X 0.233,Y -549.988,Z 918.741,A 0.000,B 0.000,C 90.000,E1 349.342} C_DIS
LIN {X 0.067,Y -556.437,Z 918.737,A 0.000,B 0.000,C 90.000,E1 348.701} C_DIS
LIN {X 0.246,Y -562.587,Z 918.733,A 0.000,B 0.000,C 90.000,E1 347.993} C_DIS
LIN {X 0.145,Y -566.149,Z 918.731,A 0.000,B 0.000,C 90.000,E1 347.589} C_DIS
LIN {X -0.067,Y -570.584,Z 918.728,A 0.000,B 0.000,C 90.000,E1 347.061} C_DIS
LIN {X -0.164,Y -577.734,Z 918.723,A 0.000,B 0.000,C 90.000,E1 346.117} C_DIS
LIN {X 0.067,Y -583.247,Z 918.718,A 0.000,B 0.000,C 90.000,E1 345.283} C_DIS
LIN {X 0.125,Y -589.236,Z 918.713,A 0.000,B 0.000,C 90.000,E1 344.338} C_DIS
LIN {X -0.152,Y -594.563,Z 918.708,A 0.000,B 0.000,C 90.000,E1 343.433} C_DIS
LIN {X 0.268,Y -598.871,Z 918.703,A 0.000,B 0.000,C 90.000,E1 342.598} C_DIS
LIN {X 0.207,Y -602.331,Z 918.700,A 0.000,B 0.000,C 90.000,E1 341.945} C_DIS
LIN {X 0.048,Y -607.571,Z 918.694,A 0.000,B 0.000,C 90.000,E1 340.913} C_DIS
LIN {X 0.015,Y -611.411,Z 918.690,A 0.000,B 0.000,C 90.000,E1 340.134} C_DIS
LIN {X 0.185,Y -616.147,Z 918.684,A 0.000,B 0.000,C 90.000,E1 339.082} C_DIS
LIN {X 0.195,Y -620.671,Z 918.678,A 0.000,B 0.000,C 90.000,E1 338.050} C_DIS
LIN {X -0.081,Y -624.897,Z 918.672,A 0.000,B 0.000,C 90.000,E1 337.050} C_DIS
LIN {X -0.061,Y -627.810,Z 918.668,A 0.000,B 0.000,C 90.000,E1 336.282} C_DIS
LIN {X -0.261,Y -630.611,Z 918.664,A 0.000,B 0.000,C 90.000,E1 335.537} C_DIS
LIN {X -0.328,Y -635.793,Z 918.656,A 0.000,B 0.000,C 90.000,E1 334.024} C_DIS
LIN {X -0.186,Y -638.271,Z 918.651,A 0.000,B 0.000,C 90.000,E1 333.256} C_DIS
LIN {X 0.105,Y -641.975,Z 918.644,A 0.000,B 0.000,C 90.000,E1 331.975} C_DIS
LIN {X 0.121,Y -644.720,Z 918.639,A 0.000,B 0.000,C 90.000,E1 330.973} C_DIS
LIN {X 0.022,Y -648.525,Z 918.631,A 0.000,B 0.000,C 90.000,E1 329.488} C_DIS
LIN {X 0.002,Y -651.446,Z 918.624,A 0.000,B 0.000,C 90.000,E1 328.250} C_DIS
LIN {X 0.153,Y -653.451,Z 918.618,A 0.000,B 0.000,C 90.000,E1 327.248} C_DIS
LIN {X -0.226,Y -655.222,Z 918.613,A 0.000,B 0.000,C 90.000,E1 326.294} C_DIS
LIN {X -0.129,Y -657.037,Z 918.606,A 0.000,B 0.000,C 90.000,E1 325.055} C_DIS
LIN {X -0.159,Y -658.629,Z 918.599,A 0.000,B 0.000,C 90.000,E1 323.829} C_DIS
LIN {X 0.373,Y -659.866,Z 918.592,A 0.000,B 0.000,C 90.000,E1 322.557} C_DIS
LIN {X 0.361,Y -660.602,Z 918.588,A 0.000,B 0.000,C 90.000,E1 321.823} C_DIS
LIN {X 0.362,Y -661.862,Z 918.580,A 0.000,B 0.000,C 90.000,E1 320.356} C_DIS
LIN {X -0.129,Y -663.038,Z 918.572,A 0.000,B 0.000,C 90.000,E1 318.933} C_DIS
LIN {X -0.183,Y -665.299,Z 918.560,A 0.000,B 0.000,C 90.000,E1 316.743} C_DIS
LIN {X 0.287,Y -665.914,Z 918.556,A 0.000,B 0.000,C 90.000,E1 315.972} C_DIS
LIN {X -0.160,Y -668.327,Z 918.539,A 0.000,B 0.000,C 90.000,E1 313.095} C_DIS
LIN {X -0.081,Y -669.748,Z 918.531,A 0.000,B 0.000,C 90.000,E1 311.634} C_DIS
LIN {X 0.017,Y -670.847,Z 918.525,A 0.000,B 0.000,C 90.000,E1 310.415} C_DIS
LIN {X -0.294,Y -672.249,Z 918.515,A 0.000,B 0.000,C 90.000,E1 308.749} C_DIS
LIN {X -0.074,Y -673.292,Z 918.507,A 0.000,B 0.000,C 90.000,E1 307.282} C_DIS
LIN {X -0.364,Y -673.721,Z 918.503,A 0.000,B 0.000,C 90.000,E1 306.583} C_DIS
LIN {X -0.383,Y -674.502,Z 918.494,A 0.000,B 0.000,C 90.000,E1 304.898} C_DIS
LIN {X -0.229,Y -675.412,Z 918.483,A 0.000,B 0.000,C 90.000,E1 302.959} C_DIS
LIN {X 0.150,Y -676.617,Z 918.472,A 0.000,B 0.000,C 90.000,E1 301.003} C_DIS
LIN {X -0.014,Y -679.554,Z 918.455,A 0.000,B 0.000,C 90.000,E1 297.897} C_DIS
LIN {X 0.285,Y -682.541,Z 918.443,A 0.000,B 0.000,C 90.000,E1 295.720} C_DIS
LIN {X 0.425,Y -684.257,Z 918.436,A 0.000,B 0.000,C 90.000,E1 294.515} C_DIS
LIN {X 0.097,Y -685.389,Z 918.431,A 0.000,B 0.000,C 90.000,E1 293.590} C_DIS
LIN {X -0.103,Y -685.727,Z 918.429,A 0.000,B 0.000,C 90.000,E1 293.131} C_DIS
LIN {X -0.157,Y -685.787,Z 918.427,A 0.000,B 0.000,C 90.000,E1 292.898} C_DIS
LIN {X 0.008,Y -685.584,Z 918.425,A 0.000,B 0.000,C 90.000,E1 292.408} C_DIS
LIN {X 0.221,Y -684.973,Z 918.423,A 0.000,B 0.000,C 90.000,E1 292.153} C_DIS
LIN {X -0.250,Y -683.239,Z 918.421,A 0.000,B 0.000,C 90.000,E1 291.716} C_DIS
LIN {X -0.149,Y -682.554,Z 918.420,A 0.000,B 0.000,C 90.000,E1 291.589} C_DIS
LIN {X -0.047,Y -681.530,Z 918.419,A 0.000,B 0.000,C 90.000,E1 291.461} C_DIS
LIN {X -0.197,Y -680.015,Z 918.419,A 0.000,B 0.000,C 90.000,E1 291.354} C_DIS
LIN {X 0.293,Y -676.910,Z 918.417,A 0.000,B 0.000,C 90.000,E1 291.099} C_DIS
LIN {X -0.192,Y -675.760,Z 918.417,A 0.000,B 0.000,C 90.000,E1 291.046} C_DIS
LIN {X 0.037,Y -674.134,Z 918.416,A 0.000,B 0.000,C 90.000,E1 290.918} C_DIS
LIN {X -0.197,Y -664.276,Z 918.413,A 0.000,B 0.000,C 90.000,E1 290.429} C_DIS
LIN {X 0.057,Y -662.318,Z 918.413,A 0.000,B 0.000,C 90.000,E1 290.301} C_DIS
LIN {X -0.299,Y -661.503,Z 918.412,A 0.000,B 0.000,C 90.000,E1 290.248} C_DIS
LIN {X -0.360,Y -661.478,Z 918.412,A 0.000,B 0.000,C 90.000,E1 290.248} C_DIS
LIN {X -0.352,Y -661.407,Z 918.411,A 0.000,B 0.000,C 90.000,E1 290.066} C_DIS
LIN {X -0.287,Y -662.529,Z 918.409,A 0.000,B 0.000,C 90.000,E1 289.577} C_DIS
LIN {X -0.216,Y -665.133,Z 918.405,A 0.000,B 0.000,C 90.000,E1 288.960} C_DIS
LIN {X -0.359,Y -670.178,Z 918.400,A 0.000,B 0.000,C 90.000,E1 288.000} C_DIS
LIN {X 0.271,Y -672.018,Z 918.398,A 0.000,B 0.000,C 90.000,E1 287.583} C_DIS
LIN {X 0.337,Y -674.312,Z 918.395,A 0.000,B 0.000,C 90.000,E1 287.094} C_DIS
LIN {X 0.166,Y -677.291,Z 918.391,A 0.000,B 0.000,C 90.000,E1 286.386} C_DIS
LIN {X 0.213,Y -679.632,Z 918.387,A 0.000,B 0.000,C 90.000,E1 285.662} C_DIS
LIN {X 0.098,Y -681.473,Z 918.383,A 0.000,B 0.000,C 90.000,E1 284.954} C_DIS
LIN {X 0.003,Y -683.024,Z 918.379,A 0.000,B 0.000,C 90.000,E1 284.245} C_DIS
LIN {X -0.076,Y -684.390,Z 918.375,A 0.000,B 0.000,C 90.000,E1 283.536} C_DIS
LIN {X -0.166,Y -685.819,Z 918.370,A 0.000,B 0.000,C 90.000,E1 282.591} C_DIS
LIN {X -0.207,Y -686.359,Z 918.367,A 0.000,B 0.000,C 90.000,E1 282.119} C_DIS
LIN {X 0.270,Y -686.939,Z 918.363,A 0.000,B 0.000,C 90.000,E1 281.366} C_DIS
LIN {X 0.234,Y -687.066,Z 918.361,A 0.000,B 0.000,C 90.000,E1 280.894} C_DIS
LIN {X 0.215,Y -687.052,Z 918.359,A 0.000,B 0.000,C 90.000,E1 280.658} C_DIS
LIN {X 0.050,Y -686.674,Z 918.357,A 0.000,B 0.000,C 90.000,E1 280.197} C_DIS
LIN {X 0.004,Y -685.932,Z 918.354,A 0.000,B 0.000,C 90.000,E1 279.726} C_DIS
LIN {X -0.135,Y -685.443,Z 918.353,A 0.000,B 0.000,C 90.000,E1 279.500} C_DIS
LIN {X -0.192,Y -684.037,Z 918.350,A 0.000,B 0.000,C 90.000,E1 279.029} C_DIS
LIN {X 0.309,Y -682.196,Z 918.347,A 0.000,B 0.000,C 90.000,E1 278.511} C_DIS
LIN {X 0.077,Y -678.938,Z 918.344,A 0.000,B 0.000,C 90.000,E1 277.814} C_DIS
LIN {X 0.325,Y -673.988,Z 918.338,A 0.000,B 0.000,C 90.000,E1 276.834} C_DIS
LIN {X 0.008,Y -670.543,Z 918.335,A 0.000,B 0.000,C 90.000,E1 276.258} C_DIS
LIN {X -0.248,Y -667.523,Z 918.332,A 0.000,B 0.000,C 90.000,E1 275.796} C_DIS
LIN {X 0.051,Y -663.190,Z 918.329,A 0.000,B 0.000,C 90.000,E1 275.163} C_DIS
LIN {X -0.255,Y -659.421,Z 918.326,A 0.000,B 0.000,C 90.000,E1 274.702} C_DIS
LIN {X 0.022,Y -655.360,Z 918.323,A 0.000,B 0.000,C 90.000,E1 274.188} C_DIS
LIN {X 0.318,Y -650.878,Z 918.321,A 0.000,B 0.000,C 90.000,E1 273.669} C_DIS
LIN {X -0.063,Y -644.686,Z 918.317,A 0.000,B 0.000,C 90.000,E1 273.094} C_DIS
LIN {X 0.090,Y -638.242,Z 918.314,A 0.000,B 0.000,C 90.000,E1 272.522} C_DIS
LIN {X -0.316,Y -631.161,Z 918.311,A 0.000,B 0.000,C 90.000,E1 272.007} C_DIS
LIN {X -0.271,Y -623.601,Z 918.308,A 0.000,B 0.000,C 90.000,E1 271.489} C_DIS
LIN {X -0.108,Y -617.376,Z 918.306,A 0.000,B 0.000,C 90.000,E1 271.088} C_DIS
LIN {X -0.279,Y -611.062,Z 918.304,A 0.000,B 0.000,C 90.000,E1 270.745} C_DIS
LIN {X 0.302,Y -604.258,Z 918.302,A 0.000,B 0.000,C 90.000,E1 270.344} C_DIS
LIN {X -0.047,Y -597.409,Z 918.300,A 0.000,B 0.000,C 90.000,E1 270.057} C_DIS
LIN {X -0.039,Y -590.276,Z 918.299,A 0.000,B 0.000,C 90.000,E1 269.771} C_DIS
LIN {X -0.277,Y -584.716,Z 918.298,A 0.000,B 0.000,C 90.000,E1 269.599} C_DIS
LIN {X -0.148,Y -577.258,Z 918.296,A 0.000,B 0.000,C 90.000,E1 269.370} C_DIS
LIN {X 0.245,Y -571.428,Z 918.296,A 0.000,B 0.000,C 90.000,E1 269.198} C_DIS
LIN {X 0.254,Y -564.791,Z 918.295,A 0.000,B 0.000,C 90.000,E1 269.083} C_DIS
LIN {X 0.072,Y -557.188,Z 918.295,A 0.000,B 0.000,C 90.000,E1 269.026} C_DIS
LIN {X 0.242,Y -552.203,Z 918.294,A 0.000,B 0.000,C 90.000,E1 268.969} C_DIS
LIN {X -0.083,Y -549.078,Z 918.294,A 0.000,B 0.000,C 90.000,E1 268.912} C_DIS
LIN {X 0.013,Y -547.286,Z 918.293,A 0.000,B 0.000,C 90.000,E1 268.797} C_DIS
LIN {X -0.113,Y -545.489,Z 918.293,A 0.000,B 0.000,C 90.000,E1 268.682} C_DIS
LIN {X -0.144,Y -545.451,Z 918.293,A 0.000,B 0.000,C 90.000,E1 268.682} C_DIS
LIN {X -0.261,Y -544.182,Z 918.291,A 0.000,B 0.000,C 90.000,E1 268.339} C_DIS
LIN {X 0.193,Y -543.798,Z 918.290,A 0.000,B 0.000,C 90.000,E1 268.108} C_DIS
LIN {X 0.106,Y -540.163,Z 918.268,A 0.000,B 0.000,C 90.000,E1 264.147} C_DIS
LIN {X -0.237,Y -539.147,Z 918.260,A 0.000,B 0.000,C 90.000,E1 262.761} C_DIS
LIN {X -0.067,Y -538.019,Z 918.252,A 0.000,B 0.000,C 90.000,E1 261.319} C_DIS
LIN {X 0.247,Y -536.672,Z 918.244,A 0.000,B 0.000,C 90.000,E1 259.859} C_DIS
LIN {X -0.197,Y -535.697,Z 918.239,A 0.000,B 0.000,C 90.000,E1 259.050} C_DIS
LIN {X 0.295,Y -533.227,Z 918.228,A 0.000,B 0.000,C 90.000,E1 256.992} C_DIS
LIN {X 0.168,Y -531.120,Z 918.218,A 0.000,B 0.000,C 90.000,E1 255.283} C_DIS
LIN {X 0.147,Y -528.631,Z 918.207,A 0.000,B 0.000,C 90.000,E1 253.268} C_DIS
LIN {X 0.015,Y -527.238,Z 918.201,A 0.000,B 0.000,C 90.000,E1 252.127} C_DIS
LIN {X -0.133,Y -524.582,Z 918.190,A 0.000,B 0.000,C 90.000,E1 250.115} C_DIS
LIN {X 0.017,Y -522.709,Z 918.181,A 0.000,B 0.000,C 90.000,E1 248.646} C_DIS
LIN {X 0.120,Y -520.732,Z 918.173,A 0.000,B 0.000,C 90.000,E1 247.177} C_DIS
LIN {X -0.241,Y -519.039,Z 918.167,A 0.000,B 0.000,C 90.000,E1 246.049} C_DIS
LIN {X -0.141,Y -516.326,Z 918.157,A 0.000,B 0.000,C 90.000,E1 244.280} C_DIS
LIN {X 0.117,Y -514.542,Z 918.151,A 0.000,B 0.000,C 90.000,E1 243.076} C_DIS
LIN {X 0.120,Y -511.598,Z 918.141,A 0.000,B 0.000,C 90.000,E1 241.307} C_DIS
LIN {X 0.062,Y -508.387,Z 918.131,A 0.000,B 0.000,C 90.000,E1 239.537} C_DIS
LIN {X 0.239,Y -506.282,Z 918.124,A 0.000,B 0.000,C 90.000,E1 238.329} C_DIS
LIN {X -0.043,Y -503.929,Z 918.118,A 0.000,B 0.000,C 90.000,E1 237.168} C_DIS
LIN {X -0.239,Y -501.973,Z 918.113,A 0.000,B 0.000,C 90.000,E1 236.294} C_DIS
LIN {X -0.145,Y -497.957,Z 918.103,A 0.000,B 0.000,C 90.000,E1 234.482} C_DIS
LIN {X -0.143,Y -492.659,Z 918.089,A 0.000,B 0.000,C 90.000,E1 232.065} C_DIS
LIN {X 0.249,Y -489.930,Z 918.082,A 0.000,B 0.000,C 90.000,E1 230.803} C_DIS
LIN {X 0.029,Y -485.104,Z 918.071,A 0.000,B 0.000,C 90.000,E1 228.690} C_DIS
LIN {X 0.001,Y -480.360,Z 918.059,A 0.000,B 0.000,C 90.000,E1 226.539} C_DIS
LIN {X -0.068,Y -476.942,Z 918.050,A 0.000,B 0.000,C 90.000,E1 225.000} C_DIS
LIN {X -0.103,Y -472.708,Z 918.040,A 0.000,B 0.000,C 90.000,E1 223.137} C_DIS
LIN {X 0.052,Y -469.179,Z 918.031,A 0.000,B 0.000,C 90.000,E1 221.553} C_DIS
LIN {X 0.016,Y -463.725,Z 918.017,A 0.000,B 0.000,C 90.000,E1 219.036} C_DIS
LIN {X 0.039,Y -461.098,Z 918.010,A 0.000,B 0.000,C 90.000,E1 217.764} C_DIS
LIN {X 0.047,Y -457.644,Z 918.001,A 0.000,B 0.000,C 90.000,E1 216.171} C_DIS
LIN {X 0.087,Y -454.257,Z 917.992,A 0.000,B 0.000,C 90.000,E1 214.565} C_DIS
LIN {X -0.122,Y -452.159,Z 917.987,A 0.000,B 0.000,C 90.000,E1 213.627} C_DIS
LIN {X 0.160,Y -446.410,Z 917.972,A 0.000,B 0.000,C 90.000,E1 211.003} C_DIS
LIN {X -0.017,Y -441.420,Z 917.960,A 0.000,B 0.000,C 90.000,E1 208.743} C_DIS
LIN {X -0.056,Y -438.541,Z 917.952,A 0.000,B 0.000,C 90.000,E1 207.436} C_DIS
LIN {X -0.124,Y -434.898,Z 917.943,A 0.000,B 0.000,C 90.000,E1 205.796} C_DIS
LIN {X -0.072,Y -431.293,Z 917.934,A 0.000,B 0.000,C 90.000,E1 204.131} C_DIS
LIN {X 0.109,Y -426.196,Z 917.921,A 0.000,B 0.000,C 90.000,E1 201.770} C_DIS
LIN {X 0.056,Y -421.812,Z 917.910,A 0.000,B 0.000,C 90.000,E1 199.758} C_DIS
LIN {X -0.064,Y -417.151,Z 917.897,A 0.000,B 0.000,C 90.000,E1 197.402} C_DIS
LIN {X 0.184,Y -413.804,Z 917.887,A 0.000,B 0.000,C 90.000,E1 195.662} C_DIS
LIN {X -0.135,Y -409.593,Z 917.876,A 0.000,B 0.000,C 90.000,E1 193.647} C_DIS
LIN {X 0.145,Y -405.438,Z 917.864,A 0.000,B 0.000,C 90.000,E1 191.535} C_DIS
LIN {X 0.170,Y -401.319,Z 917.853,A 0.000,B 0.000,C 90.000,E1 189.443} C_DIS
LIN {X 0.096,Y -397.146,Z 917.841,A 0.000,B 0.000,C 90.000,E1 187.352} C_DIS
LIN {X 0.123,Y -392.410,Z 917.827,A 0.000,B 0.000,C 90.000,E1 184.878} C_DIS
LIN {X 0.083,Y -388.672,Z 917.815,A 0.000,B 0.000,C 90.000,E1 182.751} C_DIS
LIN {X 0.011,Y -385.660,Z 917.805,A 0.000,B 0.000,C 90.000,E1 180.974} C_DIS
LIN {X -0.162,Y -379.420,Z 917.781,A 0.000,B 0.000,C 90.000,E1 176.674} C_DIS
LIN {X -0.016,Y -378.762,Z 917.777,A 0.000,B 0.000,C 90.000,E1 175.927} C_DIS
LIN {X 0.055,Y -378.338,Z 917.772,A 0.000,B 0.000,C 90.000,E1 175.008} C_DIS
LIN {X -0.118,Y -378.528,Z 917.769,A 0.000,B 0.000,C 90.000,E1 174.489} C_DIS
LIN {X 0.188,Y -378.499,Z 917.768,A 0.000,B 0.000,C 90.000,E1 174.261} C_DIS
LIN {X 0.106,Y -379.351,Z 917.764,A 0.000,B 0.000,C 90.000,E1 173.514} C_DIS
LIN {X -0.089,Y -381.047,Z 917.760,A 0.000,B 0.000,C 90.000,E1 172.818} C_DIS
LIN {X -0.149,Y -382.735,Z 917.758,A 0.000,B 0.000,C 90.000,E1 172.413} C_DIS
LIN {X -0.163,Y -385.816,Z 917.755,A 0.000,B 0.000,C 90.000,E1 171.894} C_DIS
LIN {X -0.019,Y -391.702,Z 917.751,A 0.000,B 0.000,C 90.000,E1 171.197} C_DIS
LIN {X -0.141,Y -398.745,Z 917.748,A 0.000,B 0.000,C 90.000,E1 170.622} C_DIS
LIN {X -0.107,Y -416.301,Z 917.741,A 0.000,B 0.000,C 90.000,E1 169.398} C_DIS
LIN {X 0.095,Y -422.625,Z 917.739,A 0.000,B 0.000,C 90.000,E1 168.926} C_DIS
LIN {X 0.020,Y -430.603,Z 917.735,A 0.000,B 0.000,C 90.000,E1 168.342} C_DIS
LIN {X 0.002,Y -441.372,Z 917.730,A 0.000,B 0.000,C 90.000,E1 167.465} C_DIS
LIN {X 0.028,Y -447.356,Z 917.727,A 0.000,B 0.000,C 90.000,E1 166.937} C_DIS
LIN {X 0.004,Y -457.832,Z 917.722,A 0.000,B 0.000,C 90.000,E1 165.992} C_DIS
LIN {X 0.163,Y -466.128,Z 917.717,A 0.000,B 0.000,C 90.000,E1 165.117} C_DIS
LIN {X 0.073,Y -473.180,Z 917.713,A 0.000,B 0.000,C 90.000,E1 164.393} C_DIS
LIN {X -0.210,Y -483.259,Z 917.707,A 0.000,B 0.000,C 90.000,E1 163.268} C_DIS
LIN {X 0.152,Y -490.637,Z 917.702,A 0.000,B 0.000,C 90.000,E1 162.308} C_DIS
LIN {X 0.147,Y -499.686,Z 917.695,A 0.000,B 0.000,C 90.000,E1 161.094} C_DIS
LIN {X -0.085,Y -510.332,Z 917.687,A 0.000,B 0.000,C 90.000,E1 159.625} C_DIS
LIN {X 0.075,Y -516.437,Z 917.682,A 0.000,B 0.000,C 90.000,E1 158.720} C_DIS
LIN {X -0.003,Y -525.077,Z 917.675,A 0.000,B 0.000,C 90.000,E1 157.411} C_DIS
LIN {X -0.080,Y -534.298,Z 917.667,A 0.000,B 0.000,C 90.000,E1 155.973} C_DIS
LIN {X -0.170,Y -541.355,Z 917.660,A 0.000,B 0.000,C 90.000,E1 154.845} C_DIS
LIN {X -0.206,Y -544.771,Z 917.657,A 0.000,B 0.000,C 90.000,E1 154.280} C_DIS
LIN {X -0.200,Y -552.869,Z 917.649,A 0.000,B 0.000,C 90.000,E1 152.871} C_DIS
LIN {X -0.014,Y -556.640,Z 917.645,A 0.000,B 0.000,C 90.000,E1 152.153} C_DIS
LIN {X 0.048,Y -559.717,Z 917.642,A 0.000,B 0.000,C 90.000,E1 151.591} C_DIS
LIN {X 0.180,Y -565.898,Z 917.635,A 0.000,B 0.000,C 90.000,E1 150.333} C_DIS
LIN {X 0.016,Y -571.170,Z 917.629,A 0.000,B 0.000,C 90.000,E1 149.253} C_DIS
LIN {X 0.176,Y -578.089,Z 917.621,A 0.000,B 0.000,C 90.000,E1 147.740} C_DIS
LIN {X -0.237,Y -582.183,Z 917.616,A 0.000,B 0.000,C 90.000,E1 146.834} C_DIS
LIN {X 0.141,Y -586.818,Z 917.610,A 0.000,B 0.000,C 90.000,E1 145.722} C_DIS
LIN {X -0.235,Y -591.279,Z 917.604,A 0.000,B 0.000,C 90.000,E1 144.689} C_DIS
LIN {X -0.212,Y -595.539,Z 917.598,A 0.000,B 0.000,C 90.000,E1 143.623} C_DIS
LIN {X 0.108,Y -600.567,Z 917.591,A 0.000,B 0.000,C 90.000,E1 142.271} C_DIS
LIN {X 0.157,Y -609.933,Z 917.577,A 0.000,B 0.000,C 90.000,E1 139.908} C_DIS
LIN {X -0.001,Y -616.195,Z 917.569,A 0.000,B 0.000,C 90.000,E1 138.366} C_DIS
LIN {X 0.120,Y -621.420,Z 917.562,A 0.000,B 0.000,C 90.000,E1 137.067} C_DIS
LIN {X -0.264,Y -627.882,Z 917.553,A 0.000,B 0.000,C 90.000,E1 135.567} C_DIS
LIN {X 0.140,Y -632.015,Z 917.547,A 0.000,B 0.000,C 90.000,E1 134.514} C_DIS
LIN {X 0.063,Y -637.160,Z 917.540,A 0.000,B 0.000,C 90.000,E1 133.257} C_DIS
LIN {X 0.072,Y -642.188,Z 917.533,A 0.000,B 0.000,C 90.000,E1 132.000} C_DIS
LIN {X 0.080,Y -649.092,Z 917.524,A 0.000,B 0.000,C 90.000,E1 130.253} C_DIS
LIN {X -0.159,Y -653.850,Z 917.517,A 0.000,B 0.000,C 90.000,E1 129.036} C_DIS
LIN {X -0.229,Y -658.578,Z 917.510,A 0.000,B 0.000,C 90.000,E1 127.810} C_DIS
LIN {X -0.217,Y -663.157,Z 917.503,A 0.000,B 0.000,C 90.000,E1 126.583} C_DIS
LIN {X -0.098,Y -666.694,Z 917.498,A 0.000,B 0.000,C 90.000,E1 125.598} C_DIS
LIN {X 0.070,Y -670.101,Z 917.492,A 0.000,B 0.000,C 90.000,E1 124.612} C_DIS
LIN {X -0.244,Y -672.529,Z 917.488,A 0.000,B 0.000,C 90.000,E1 123.913} C_DIS
LIN {X 0.024,Y -674.741,Z 917.484,A 0.000,B 0.000,C 90.000,E1 123.166} C_DIS
LIN {X -0.083,Y -677.486,Z 917.479,A 0.000,B 0.000,C 90.000,E1 122.212} C_DIS
LIN {X 0.237,Y -679.305,Z 917.475,A 0.000,B 0.000,C 90.000,E1 121.465} C_DIS
LIN {X 0.377,Y -681.977,Z 917.468,A 0.000,B 0.000,C 90.000,E1 120.256} C_DIS
LIN {X -0.202,Y -683.331,Z 917.464,A 0.000,B 0.000,C 90.000,E1 119.589} C_DIS
LIN {X 0.252,Y -685.274,Z 917.458,A 0.000,B 0.000,C 90.000,E1 118.359} C_DIS
LIN {X 0.082,Y -685.941,Z 917.455,A 0.000,B 0.000,C 90.000,E1 117.897} C_DIS
LIN {X 0.045,Y -686.797,Z 917.450,A 0.000,B 0.000,C 90.000,E1 116.950} C_DIS
LIN {X 0.107,Y -687.129,Z 917.446,A 0.000,B 0.000,C 90.000,E1 116.232} C_DIS
LIN {X 0.093,Y -687.385,Z 917.441,A 0.000,B 0.000,C 90.000,E1 115.283} C_DIS
LIN {X 0.084,Y -687.275,Z 917.435,A 0.000,B 0.000,C 90.000,E1 114.335} C_DIS
LIN {X -0.375,Y -687.016,Z 917.433,A 0.000,B 0.000,C 90.000,E1 113.898} C_DIS
LIN {X -0.153,Y -686.838,Z 917.431,A 0.000,B 0.000,C 90.000,E1 113.643} C_DIS
LIN {X 0.016,Y -685.981,Z 917.429,A 0.000,B 0.000,C 90.000,E1 113.153} C_DIS
LIN {X 0.235,Y -685.430,Z 917.427,A 0.000,B 0.000,C 90.000,E1 112.898} C_DIS
LIN {X -0.183,Y -684.136,Z 917.426,A 0.000,B 0.000,C 90.000,E1 112.695} C_DIS
LIN {X -0.095,Y -681.621,Z 917.424,A 0.000,B 0.000,C 90.000,E1 112.259} C_DIS
LIN {X -0.252,Y -680.421,Z 917.423,A 0.000,B 0.000,C 90.000,E1 112.153} C_DIS
LIN {X 0.207,Y -677.118,Z 917.422,A 0.000,B 0.000,C 90.000,E1 111.897} C_DIS
LIN {X -0.314,Y -675.371,Z 917.421,A 0.000,B 0.000,C 90.000,E1 111.844} C_DIS
LIN {X -0.205,Y -671.759,Z 917.420,A 0.000,B 0.000,C 90.000,E1 111.663} C_DIS
LIN {X -0.224,Y -669.690,Z 917.420,A 0.000,B 0.000,C 90.000,E1 111.589} C_DIS
LIN {X -0.088,Y -664.356,Z 917.419,A 0.000,B 0.000,C 90.000,E1 111.461} C_DIS
LIN {X 0.066,Y -662.092,Z 917.419,A 0.000,B 0.000,C 90.000,E1 111.408} C_DIS
LIN {X -0.302,Y -659.117,Z 917.419,A 0.000,B 0.000,C 90.000,E1 111.408} C_DIS
LIN {X -0.232,Y -649.942,Z 917.419,A 0.000,B 0.000,C 90.000,E1 111.354} C_DIS
LIN {X 0.260,Y -641.992,Z 917.418,A 0.000,B 0.000,C 90.000,E1 111.280} C_DIS
LIN {X -0.037,Y -638.527,Z 917.418,A 0.000,B 0.000,C 90.000,E1 111.280} C_DIS
LIN {X -0.276,Y -632.835,Z 917.418,A 0.000,B 0.000,C 90.000,E1 111.227} C_DIS
LIN {X -0.017,Y -626.797,Z 917.417,A 0.000,B 0.000,C 90.000,E1 111.099} C_DIS
LIN {X -0.064,Y -621.231,Z 917.417,A 0.000,B 0.000,C 90.000,E1 110.972} C_DIS
LIN {X 0.066,Y -613.851,Z 917.415,A 0.000,B 0.000,C 90.000,E1 110.737} C_DIS
LIN {X -0.317,Y -605.274,Z 917.413,A 0.000,B 0.000,C 90.000,E1 110.429} C_DIS
LIN {X 0.214,Y -599.034,Z 917.412,A 0.000,B 0.000,C 90.000,E1 110.066} C_DIS
LIN {X 0.130,Y -588.350,Z 917.408,A 0.000,B 0.000,C 90.000,E1 109.396} C_DIS
LIN {X -0.145,Y -579.340,Z 917.405,A 0.000,B 0.000,C 90.000,E1 108.833} C_DIS
LIN {X -0.118,Y -572.463,Z 917.403,A 0.000,B 0.000,C 90.000,E1 108.471} C_DIS
LIN {X 0.189,Y -565.333,Z 917.401,A 0.000,B 0.000,C 90.000,E1 108.127} C_DIS
LIN {X -0.111,Y -556.867,Z 917.399,A 0.000,B 0.000,C 90.000,E1 107.819} C_DIS
LIN {X -0.090,Y -555.794,Z 917.399,A 0.000,B 0.000,C 90.000,E1 107.764} C_DIS
LIN {X 0.126,Y -554.507,Z 917.398,A 0.000,B 0.000,C 90.000,E1 107.638} C_DIS
LIN {X -0.004,Y -553.793,Z 917.398,A 0.000,B 0.000,C 90.000,E1 107.583} C_DIS
LIN {X -0.042,Y -553.757,Z 917.398,A 0.000,B 0.000,C 90.000,E1 107.583} C_DIS
LIN {X -0.068,Y -553.493,Z 917.397,A 0.000,B 0.000,C 90.000,E1 107.402} C_DIS
LIN {X 0.055,Y -553.544,Z 917.392,A 0.000,B 0.000,C 90.000,E1 106.551} C_DIS
LIN {X -0.284,Y -554.134,Z 917.384,A 0.000,B 0.000,C 90.000,E1 105.190} C_DIS
LIN {X -0.100,Y -555.215,Z 917.372,A 0.000,B 0.000,C 90.000,E1 102.939} C_DIS
LIN {X -0.141,Y -556.726,Z 917.359,A 0.000,B 0.000,C 90.000,E1 100.715} C_DIS
LIN {X 0.027,Y -557.974,Z 917.350,A 0.000,B 0.000,C 90.000,E1 99.029} C_DIS
LIN {X 0.205,Y -559.376,Z 917.339,A 0.000,B 0.000,C 90.000,E1 97.068} C_DIS
LIN {X -0.214,Y -560.347,Z 917.330,A 0.000,B 0.000,C 90.000,E1 95.448} C_DIS
LIN {X 0.170,Y -560.975,Z 917.324,A 0.000,B 0.000,C 90.000,E1 94.302} C_DIS
LIN {X 0.234,Y -561.806,Z 917.315,A 0.000,B 0.000,C 90.000,E1 92.636} C_DIS
LIN {X 0.182,Y -562.390,Z 917.307,A 0.000,B 0.000,C 90.000,E1 91.260} C_DIS
LIN {X 0.027,Y -562.778,Z 917.301,A 0.000,B 0.000,C 90.000,E1 90.172} C_DIS
LIN {X 0.083,Y -563.133,Z 917.292,A 0.000,B 0.000,C 90.000,E1 88.511} C_DIS
LIN {X 0.153,Y -563.504,Z 917.283,A 0.000,B 0.000,C 90.000,E1 86.849} C_DIS
LIN {X -0.303,Y -563.763,Z 917.273,A 0.000,B 0.000,C 90.000,E1 85.241} C_DIS
LIN {X 0.012,Y -564.080,Z 917.263,A 0.000,B 0.000,C 90.000,E1 83.280} C_DIS
LIN {X 0.258,Y -564.433,Z 917.254,A 0.000,B 0.000,C 90.000,E1 81.602} C_DIS
LIN {X -0.218,Y -564.886,Z 917.246,A 0.000,B 0.000,C 90.000,E1 80.274} C_DIS
LIN {X -0.151,Y -565.726,Z 917.235,A 0.000,B 0.000,C 90.000,E1 78.342} C_DIS
LIN {X -0.057,Y -566.800,Z 917.224,A 0.000,B 0.000,C 90.000,E1 76.408} C_DIS
LIN {X -0.158,Y -567.591,Z 917.217,A 0.000,B 0.000,C 90.000,E1 75.046} C_DIS
LIN {X 0.079,Y -568.461,Z 917.208,A 0.000,B 0.000,C 90.000,E1 73.378} C_DIS
LIN {X -0.218,Y -569.156,Z 917.199,A 0.000,B 0.000,C 90.000,E1 71.764} C_DIS
LIN {X -0.141,Y -569.752,Z 917.190,A 0.000,B 0.000,C 90.000,E1 70.115} C_DIS
LIN {X -0.045,Y -570.167,Z 917.180,A 0.000,B 0.000,C 90.000,E1 68.465} C_DIS
LIN {X -0.088,Y -570.441,Z 917.173,A 0.000,B 0.000,C 90.000,E1 67.102} C_DIS
LIN {X -0.304,Y -570.634,Z 917.164,A 0.000,B 0.000,C 90.000,E1 65.485} C_DIS
LIN {X 0.049,Y -570.715,Z 917.158,A 0.000,B 0.000,C 90.000,E1 64.357} C_DIS
LIN {X -0.030,Y -570.790,Z 917.150,A 0.000,B 0.000,C 90.000,E1 62.999} C_DIS
LIN {X -0.102,Y -570.755,Z 917.142,A 0.000,B 0.000,C 90.000,E1 61.641} C_DIS
LIN {X 0.101,Y -570.736,Z 917.135,A 0.000,B 0.000,C 90.000,E1 60.255} C_DIS
LIN {X -0.303,Y -570.569,Z 917.129,A 0.000,B 0.000,C 90.000,E1 59.203} C_DIS
LIN {X 0.245,Y -570.464,Z 917.124,A 0.000,B 0.000,C 90.000,E1 58.329} C_DIS
LIN {X -0.059,Y -569.857,Z 917.117,A 0.000,B 0.000,C 90.000,E1 56.993} C_DIS
LIN {X 0.248,Y -569.168,Z 917.109,A 0.000,B 0.000,C 90.000,E1 55.595} C_DIS
LIN {X -0.041,Y -568.450,Z 917.103,A 0.000,B 0.000,C 90.000,E1 54.529} C_DIS
LIN {X 0.122,Y -567.433,Z 917.097,A 0.000,B 0.000,C 90.000,E1 53.417} C_DIS
LIN {X -0.193,Y -566.188,Z 917.091,A 0.000,B 0.000,C 90.000,E1 52.351} C_DIS
LIN {X -0.181,Y -564.797,Z 917.085,A 0.000,B 0.000,C 90.000,E1 51.251} C_DIS
LIN {X -0.189,Y -563.039,Z 917.079,A 0.000,B 0.000,C 90.000,E1 50.150} C_DIS
LIN {X 0.043,Y -561.573,Z 917.074,A 0.000,B 0.000,C 90.000,E1 49.299} C_DIS
LIN {X -0.194,Y -560.514,Z 917.071,A 0.000,B 0.000,C 90.000,E1 48.771} C_DIS
LIN {X 0.095,Y -557.980,Z 917.065,A 0.000,B 0.000,C 90.000,E1 47.634} C_DIS
LIN {X 0.207,Y -556.587,Z 917.062,A 0.000,B 0.000,C 90.000,E1 47.067} C_DIS
LIN {X -0.069,Y -555.039,Z 917.059,A 0.000,B 0.000,C 90.000,E1 46.539} C_DIS
LIN {X -0.322,Y -552.447,Z 917.054,A 0.000,B 0.000,C 90.000,E1 45.729} C_DIS
LIN {X -0.243,Y -550.575,Z 917.051,A 0.000,B 0.000,C 90.000,E1 45.162} C_DIS
LIN {X 0.237,Y -547.399,Z 917.046,A 0.000,B 0.000,C 90.000,E1 44.271} C_DIS
LIN {X 0.277,Y -545.149,Z 917.043,A 0.000,B 0.000,C 90.000,E1 43.704} C_DIS
LIN {X 0.122,Y -542.063,Z 917.039,A 0.000,B 0.000,C 90.000,E1 43.014} C_DIS
LIN {X -0.270,Y -536.515,Z 917.033,A 0.000,B 0.000,C 90.000,E1 41.919} C_DIS
LIN {X 0.254,Y -532.613,Z 917.029,A 0.000,B 0.000,C 90.000,E1 41.148} C_DIS
LIN {X -0.014,Y -528.377,Z 917.025,A 0.000,B 0.000,C 90.000,E1 40.458} C_DIS
LIN {X 0.086,Y -523.806,Z 917.021,A 0.000,B 0.000,C 90.000,E1 39.725} C_DIS
LIN {X 0.143,Y -519.030,Z 917.017,A 0.000,B 0.000,C 90.000,E1 38.991} C_DIS
LIN {X 0.158,Y -513.880,Z 917.013,A 0.000,B 0.000,C 90.000,E1 38.257} C_DIS
LIN {X 0.011,Y -509.574,Z 917.009,A 0.000,B 0.000,C 90.000,E1 37.684} C_DIS
LIN {X 0.109,Y -506.295,Z 917.007,A 0.000,B 0.000,C 90.000,E1 37.237} C_DIS
LIN {X 0.135,Y -500.367,Z 917.003,A 0.000,B 0.000,C 90.000,E1 36.503} C_DIS
LIN {X 0.173,Y -498.055,Z 917.001,A 0.000,B 0.000,C 90.000,E1 36.217} C_DIS
LIN {X 0.270,Y -490.058,Z 916.996,A 0.000,B 0.000,C 90.000,E1 35.311} C_DIS
LIN {X 0.138,Y -483.022,Z 916.992,A 0.000,B 0.000,C 90.000,E1 34.612} C_DIS
LIN {X 0.068,Y -477.263,Z 916.989,A 0.000,B 0.000,C 90.000,E1 34.072} C_DIS
LIN {X -0.246,Y -466.922,Z 916.984,A 0.000,B 0.000,C 90.000,E1 33.166} C_DIS
LIN {X -0.159,Y -460.861,Z 916.981,A 0.000,B 0.000,C 90.000,E1 32.625} C_DIS
LIN {X -0.118,Y -447.172,Z 916.975,A 0.000,B 0.000,C 90.000,E1 31.465} C_DIS
LIN {X 0.050,Y -433.204,Z 916.968,A 0.000,B 0.000,C 90.000,E1 30.285} C_DIS
LIN {X -0.148,Y -413.443,Z 916.959,A 0.000,B 0.000,C 90.000,E1 28.565} C_DIS
LIN {X 0.128,Y -400.286,Z 916.952,A 0.000,B 0.000,C 90.000,E1 27.257} C_DIS
LIN {X -0.058,Y -396.242,Z 916.949,A 0.000,B 0.000,C 90.000,E1 26.821} C_DIS
LIN {X 0.003,Y -392.485,Z 916.946,A 0.000,B 0.000,C 90.000,E1 26.283} C_DIS
LIN {X -0.043,Y -390.688,Z 916.944,A 0.000,B 0.000,C 90.000,E1 25.848} C_DIS
LIN {X -0.078,Y -390.077,Z 916.943,A 0.000,B 0.000,C 90.000,E1 25.720} C_DIS
LIN {X 0.163,Y -389.408,Z 916.941,A 0.000,B 0.000,C 90.000,E1 25.283} C_DIS
LIN {X -0.177,Y -388.992,Z 916.940,A 0.000,B 0.000,C 90.000,E1 25.155} C_DIS
LIN {X 0.220,Y -388.524,Z 916.936,A 0.000,B 0.000,C 90.000,E1 24.387} C_DIS
LIN {X 0.095,Y -389.028,Z 916.930,A 0.000,B 0.000,C 90.000,E1 23.334} C_DIS
LIN {X -0.133,Y -392.733,Z 916.908,A 0.000,B 0.000,C 90.000,E1 19.450} C_DIS
LIN {X -0.109,Y -396.477,Z 916.890,A 0.000,B 0.000,C 90.000,E1 16.260} C_DIS
LIN {X 0.110,Y -400.626,Z 916.873,A 0.000,B 0.000,C 90.000,E1 13.063} C_DIS
LIN {X -0.180,Y -404.252,Z 916.859,A 0.000,B 0.000,C 90.000,E1 10.658} C_DIS
LIN {X -0.147,Y -409.428,Z 916.842,A 0.000,B 0.000,C 90.000,E1 7.530} C_DIS
LIN {X -0.018,Y -415.156,Z 916.825,A 0.000,B 0.000,C 90.000,E1 4.416} C_DIS
LIN {X 0.145,Y -420.105,Z 916.811,A 0.000,B 0.000,C 90.000,E1 2.007} C_DIS
LIN {X -0.212,Y -426.060,Z 916.797,A 0.000,B 0.000,C 90.000,E1 359.484} C_DIS
LIN {X 0.107,Y -430.361,Z 916.788,A 0.000,B 0.000,C 90.000,E1 357.764} C_DIS
LIN {X -0.217,Y -431.954,Z 916.785,A 0.000,B 0.000,C 90.000,E1 357.306} C_DIS
LIN {X -0.141,Y -433.248,Z 916.783,A 0.000,B 0.000,C 90.000,E1 356.963} C_DIS
LIN {X 0.040,Y -435.230,Z 916.781,A 0.000,B 0.000,C 90.000,E1 356.560} C_DIS
LIN {X -0.112,Y -436.774,Z 916.780,A 0.000,B 0.000,C 90.000,E1 356.331} C_DIS
LIN {X 0.069,Y -442.189,Z 916.777,A 0.000,B 0.000,C 90.000,E1 355.812} C_DIS
LIN {X -0.081,Y -447.386,Z 916.775,A 0.000,B 0.000,C 90.000,E1 355.527} C_DIS
LIN {X -0.108,Y -458.836,Z 916.772,A 0.000,B 0.000,C 90.000,E1 355.008} C_DIS
LIN {X -0.111,Y -468.516,Z 916.770,A 0.000,B 0.000,C 90.000,E1 354.546} C_DIS
LIN {X 0.039,Y -481.862,Z 916.766,A 0.000,B 0.000,C 90.000,E1 353.856} C_DIS
LIN {X 0.044,Y -491.511,Z 916.763,A 0.000,B 0.000,C 90.000,E1 353.337} C_DIS
LIN {X 0.028,Y -502.879,Z 916.760,A 0.000,B 0.000,C 90.000,E1 352.704} C_DIS
LIN {X -0.013,Y -510.955,Z 916.757,A 0.000,B 0.000,C 90.000,E1 352.243} C_DIS
LIN {X -0.111,Y -520.417,Z 916.754,A 0.000,B 0.000,C 90.000,E1 351.659} C_DIS
LIN {X -0.162,Y -529.478,Z 916.750,A 0.000,B 0.000,C 90.000,E1 351.027} C_DIS
LIN {X 0.047,Y -535.565,Z 916.748,A 0.000,B 0.000,C 90.000,E1 350.557} C_DIS
LIN {X -0.074,Y -543.904,Z 916.744,A 0.000,B 0.000,C 90.000,E1 349.859} C_DIS
LIN {X -0.020,Y -550.656,Z 916.740,A 0.000,B 0.000,C 90.000,E1 349.218} C_DIS
LIN {X -0.179,Y -557.114,Z 916.737,A 0.000,B 0.000,C 90.000,E1 348.578} C_DIS
LIN {X -0.025,Y -564.248,Z 916.732,A 0.000,B 0.000,C 90.000,E1 347.757} C_DIS
LIN {X -0.070,Y -570.966,Z 916.727,A 0.000,B 0.000,C 90.000,E1 346.937} C_DIS
LIN {X -0.158,Y -578.105,Z 916.722,A 0.000,B 0.000,C 90.000,E1 345.992} C_DIS
LIN {X -0.068,Y -583.626,Z 916.718,A 0.000,B 0.000,C 90.000,E1 345.172} C_DIS
LIN {X 0.149,Y -589.582,Z 916.712,A 0.000,B 0.000,C 90.000,E1 344.212} C_DIS
LIN {X -0.290,Y -594.955,Z 916.707,A 0.000,B 0.000,C 90.000,E1 343.323} C_DIS
LIN {X -0.208,Y -598.567,Z 916.704,A 0.000,B 0.000,C 90.000,E1 342.653} C_DIS
LIN {X -0.031,Y -604.031,Z 916.698,A 0.000,B 0.000,C 90.000,E1 341.583} C_DIS
LIN {X 0.139,Y -607.330,Z 916.694,A 0.000,B 0.000,C 90.000,E1 340.913} C_DIS
LIN {X 0.076,Y -611.790,Z 916.689,A 0.000,B 0.000,C 90.000,E1 340.007} C_DIS
LIN {X 0.001,Y -617.712,Z 916.682,A 0.000,B 0.000,C 90.000,E1 338.720} C_DIS
LIN {X 0.261,Y -622.143,Z 916.676,A 0.000,B 0.000,C 90.000,E1 337.667} C_DIS
LIN {X 0.010,Y -626.281,Z 916.670,A 0.000,B 0.000,C 90.000,E1 336.666} C_DIS
LIN {X -0.187,Y -630.085,Z 916.665,A 0.000,B 0.000,C 90.000,E1 335.665} C_DIS
LIN {X -0.303,Y -634.477,Z 916.658,A 0.000,B 0.000,C 90.000,E1 334.409} C_DIS
SetRPM(0)
End
